LIN {X 0,Y 254.249,Z 344.944,A -85,B 0,C 180,E1 -18935.484,E2 -18935.484} C_VEL
LIN {X 0,Y 252.335,Z 350.692,A -85,B 0,C 180,E1 -18937.788,E2 -18937.788} C_VEL
LIN {X 0,Y 250.743,Z 355.289,A -85,B 0,C 180,E1 -18940.14,E2 -18940.14} C_VEL
LIN {X 0,Y 249.286,Z 359.262,A -85,B 0,C 180,E1 -18942.862,E2 -18942.862} C_VEL
LIN {X 0,Y 248.38,Z 361.475,A -85,B 0,C 180,E1 -18945.022,E2 -18945.022} C_VEL
LIN {X 0,Y 247.644,Z 363.12,A -85,B 0,C 180,E1 -18947.549,E2 -18947.549} C_VEL
LIN {X 0,Y 247.177,Z 363.796,A -85,B 0,C 180,E1 -18950.147,E2 -18950.147} C_VEL
LIN {X 0,Y 246.95,Z 363.273,A -85,B 0,C 180,E1 -18953.299,E2 -18953.299} C_VEL
LIN {X 0,Y 247.021,Z 361.92,A -85,B 0,C 180,E1 -18955.596,E2 -18955.596} C_VEL
LIN {X 0,Y 247.445,Z 359.132,A -85,B 0,C 180,E1 -18958.437,E2 -18958.437} C_VEL
LIN {X 0,Y 248.133,Z 354.726,A -85,B 0,C 180,E1 -18961.405,E2 -18961.405} C_VEL
LIN {X 0,Y 248.912,Z 349.759,A -85,B 0,C 180,E1 -18963.884,E2 -18963.884} C_VEL
LIN {X 0,Y 250.067,Z 343.333,A -85,B 0,C 180,E1 -18966.392,E2 -18966.392} C_VEL
LIN {X 0,Y 251.344,Z 335.987,A -85,B 0,C 180,E1 -18968.685,E2 -18968.685} C_VEL
LIN {X 0,Y 253.013,Z 326.632,A -85,B 0,C 180,E1 -18971.005,E2 -18971.005} C_VEL
LIN {X 0,Y 254.61,Z 316.87,A -85,B 0,C 180,E1 -18972.946,E2 -18972.946} C_VEL
LIN {X 0,Y 256.282,Z 305.858,A -85,B 0,C 180,E1 -18974.696,E2 -18974.696} C_VEL
LIN {X 0,Y 257.875,Z 293.608,A -85,B 0,C 180,E1 -18976.204,E2 -18976.204} C_VEL
LIN {X 0,Y 259.117,Z 281.075,A -85,B 0,C 180,E1 -18977.388,E2 -18977.388} C_VEL
LIN {X 0,Y 260.143,Z 267.516,A -85,B 0,C 180,E1 -18978.285,E2 -18978.285} C_VEL
LIN {X 0,Y 260.78,Z 254.66,A -85,B 0,C 180,E1 -18978.831,E2 -18978.831} C_VEL
LIN {X 0,Y 263.039,Z 190.676,A -85,B 0,C 180,E1 -18980.701,E2 -18980.701} C_VEL
LIN {X 0,Y 258.834,Z 179.431,A -85,B 0,C 180,E1 -18981.466,E2 -18981.466} C_VEL
LIN {X 0,Y 250.247,Z 159.861,A -85,B 0,C 180,E1 -18982.993,E2 -18982.993} C_VEL
LIN {X 0,Y 249.456,Z 157.414,A -85,B 0,C 180,E1 -18983.174,E2 -18983.174} C_VEL
LIN {X 0,Y 249.675,Z 157.384,A -85,B 0,C 180,E1 -18988.387,E2 -18988.387} C_VEL
LIN {X 0,Y 249.675,Z 157.386,A -85,B 0,C 180,E1 -18991.613,E2 -18991.613} C_VEL
LIN {X 0,Y 249.431,Z 157.415,A -85,B 0,C 180,E1 -18996.471,E2 -18996.471} C_VEL
LIN {X 0,Y 249.342,Z 157.425,A -85,B 0,C 180,E1 -18999.736,E2 -18999.736} C_VEL
LIN {X 0,Y 249.175,Z 157.448,A -85,B 0,C 180,E1 -19004.705,E2 -19004.705} C_VEL
LIN {X 0,Y 249.108,Z 157.452,A -85,B 0,C 180,E1 -19008.08,E2 -19008.08} C_VEL
LIN {X 0,Y 249.08,Z 157.456,A -85,B 0,C 180,E1 -19011.519,E2 -19011.519} C_VEL
LIN {X 0,Y 249.117,Z 157.452,A -85,B 0,C 180,E1 -19015.476,E2 -19015.476} C_VEL
LIN {X 0,Y 249.083,Z 157.458,A -85,B 0,C 180,E1 -19018.994,E2 -19018.994} C_VEL
LIN {X 0,Y 249.033,Z 157.465,A -85,B 0,C 180,E1 -19022.425,E2 -19022.425} C_VEL
LIN {X 0,Y 249.056,Z 157.462,A -85,B 0,C 180,E1 -19026.341,E2 -19026.341} C_VEL
LIN {X 0,Y 249.005,Z 157.462,A -85,B 0,C 180,E1 -19030.478,E2 -19030.478} C_VEL
LIN {X 0,Y 249.001,Z 157.467,A -85,B 0,C 180,E1 -19034.879,E2 -19034.879} C_VEL
LIN {X 0,Y 249.015,Z 157.463,A -85,B 0,C 180,E1 -19037.363,E2 -19037.363} C_VEL
LIN {X 0,Y 249.047,Z 157.459,A -85,B 0,C 180,E1 -19042.199,E2 -19042.199} C_VEL
LIN {X 0,Y 249.057,Z 157.461,A -85,B 0,C 180,E1 -19045.642,E2 -19045.642} C_VEL
LIN {X 0,Y 249.047,Z 157.457,A -85,B 0,C 180,E1 -19049.473,E2 -19049.473} C_VEL
LIN {X 0,Y 249.068,Z 157.454,A -85,B 0,C 180,E1 -19053.162,E2 -19053.162} C_VEL
LIN {X 0,Y 249.06,Z 157.459,A -85,B 0,C 180,E1 -19056.731,E2 -19056.731} C_VEL
LIN {X 0,Y 249.108,Z 157.448,A -85,B 0,C 180,E1 -19060.212,E2 -19060.212} C_VEL
LIN {X 0,Y 249.241,Z 157.432,A -85,B 0,C 180,E1 -19063.622,E2 -19063.622} C_VEL
LIN {X 0,Y 249.252,Z 157.435,A -85,B 0,C 180,E1 -19068.617,E2 -19068.617} C_VEL
LIN {X 0,Y 249.481,Z 157.4,A -85,B 0,C 180,E1 -19071.903,E2 -19071.903} C_VEL
LIN {X 0,Y 249.436,Z 157.41,A -85,B 0,C 180,E1 -19076.77,E2 -19076.77} C_VEL
LIN {X 0,Y 249.728,Z 157.373,A -85,B 0,C 180,E1 -19080,E2 -19080} C_VEL
LIN {X 0,Y 249.435,Z 157.406,A -85,B 0,C 180,E1 -19083.231,E2 -19083.231} C_VEL
LIN {X 0,Y 249.479,Z 157.406,A -85,B 0,C 180,E1 -19088.098,E2 -19088.098} C_VEL
LIN {X 0,Y 249.21,Z 157.434,A -85,B 0,C 180,E1 -19092.351,E2 -19092.351} C_VEL
LIN {X 0,Y 248.532,Z 157.522,A -85,B 0,C 180,E1 -19093.701,E2 -19093.701} C_VEL
LIN {X 0,Y 245.64,Z 157.885,A -85,B 0,C 180,E1 -19095.9,E2 -19095.9} C_VEL
LIN {X 0,Y 243.178,Z 158.191,A -85,B 0,C 180,E1 -19097.691,E2 -19097.691} C_VEL
LIN {X 0,Y 242.115,Z 158.322,A -85,B 0,C 180,E1 -19099.081,E2 -19099.081} C_VEL
LIN {X 0,Y 242.025,Z 158.331,A -85,B 0,C 180,E1 -19099.553,E2 -19099.553} C_VEL
LIN {X 0,Y 242.041,Z 158.335,A -85,B 0,C 180,E1 -19103.986,E2 -19103.986} C_VEL
LIN {X 0,Y 242.007,Z 158.336,A -85,B 0,C 180,E1 -19107.688,E2 -19107.688} C_VEL
LIN {X 0,Y 241.977,Z 158.341,A -85,B 0,C 180,E1 -19111.52,E2 -19111.52} C_VEL
LIN {X 0,Y 242.03,Z 158.336,A -85,B 0,C 180,E1 -19115.605,E2 -19115.605} C_VEL
LIN {X 0,Y 241.983,Z 158.342,A -85,B 0,C 180,E1 -19119.714,E2 -19119.714} C_VEL
LIN {X 0,Y 241.939,Z 158.349,A -85,B 0,C 180,E1 -19124.201,E2 -19124.201} C_VEL
LIN {X 0,Y 241.956,Z 158.348,A -85,B 0,C 180,E1 -19128.082,E2 -19128.082} C_VEL
LIN {X 0,Y 242.043,Z 158.414,A -85,B 0,C 180,E1 -19132.281,E2 -19132.281} C_VEL
LIN {X 0,Y 244.127,Z 167.645,A -85,B 0,C 180,E1 -19135.754,E2 -19135.754} C_VEL
LIN {X 0,Y 246.271,Z 177.912,A -85,B 0,C 180,E1 -19139.352,E2 -19139.352} C_VEL
LIN {X 0,Y 249.889,Z 188.242,A -85,B 0,C 180,E1 -19140.086,E2 -19140.086} C_VEL
LIN {X 0,Y 254.57,Z 225.349,A -85,B 0,C 180,E1 -19141.798,E2 -19141.798} C_VEL
LIN {X 0,Y 255.275,Z 233.674,A -85,B 0,C 180,E1 -19142.141,E2 -19142.141} C_VEL
LIN {X 0,Y 253.345,Z 287.616,A -85,B 0,C 180,E1 -19143.816,E2 -19143.816} C_VEL
LIN {X 0,Y 252.151,Z 301.614,A -85,B 0,C 180,E1 -19144.57,E2 -19144.57} C_VEL
LIN {X 0,Y 250.865,Z 313.126,A -85,B 0,C 180,E1 -19145.482,E2 -19145.482} C_VEL
LIN {X 0,Y 249.22,Z 324.982,A -85,B 0,C 180,E1 -19146.747,E2 -19146.747} C_VEL
LIN {X 0,Y 247.383,Z 336.431,A -85,B 0,C 180,E1 -19148.326,E2 -19148.326} C_VEL
LIN {X 0,Y 245.624,Z 346.791,A -85,B 0,C 180,E1 -19150.137,E2 -19150.137} C_VEL
LIN {X 0,Y 243.711,Z 356.55,A -85,B 0,C 180,E1 -19152.285,E2 -19152.285} C_VEL
LIN {X 0,Y 242.748,Z 363.075,A -85,B 0,C 180,E1 -19154.035,E2 -19154.035} C_VEL
LIN {X 0,Y 241.478,Z 370.708,A -85,B 0,C 180,E1 -19156.536,E2 -19156.536} C_VEL
LIN {X 0,Y 240.617,Z 376.823,A -85,B 0,C 180,E1 -19159.056,E2 -19159.056} C_VEL
LIN {X 0,Y 240.174,Z 381.638,A -85,B 0,C 180,E1 -19161.587,E2 -19161.587} C_VEL
LIN {X 0,Y 240.026,Z 385.851,A -85,B 0,C 180,E1 -19164.582,E2 -19164.582} C_VEL
LIN {X 0,Y 240.052,Z 387.865,A -85,B 0,C 180,E1 -19166.643,E2 -19166.643} C_VEL
LIN {X 0,Y 240.072,Z 389.047,A -85,B 0,C 180,E1 -19168.322,E2 -19168.322} C_VEL
LIN {X 0,Y 240.122,Z 389.77,A -85,B 0,C 180,E1 -19170,E2 -19170} C_VEL
LIN {X 0,Y 240.033,Z 390.065,A -85,B 0,C 180,E1 -19171.678,E2 -19171.678} C_VEL
LIN {X 0,Y 239.948,Z 389.962,A -85,B 0,C 180,E1 -19173.358,E2 -19173.358} C_VEL
LIN {X 0,Y 239.882,Z 389.463,A -85,B 0,C 180,E1 -19175.042,E2 -19175.042} C_VEL
LIN {X 0,Y 239.894,Z 388.533,A -85,B 0,C 180,E1 -19176.73,E2 -19176.73} C_VEL
LIN {X 0,Y 240.123,Z 387.193,A -85,B 0,C 180,E1 -19178.415,E2 -19178.415} C_VEL
LIN {X 0,Y 240.68,Z 384.41,A -85,B 0,C 180,E1 -19180.941,E2 -19180.941} C_VEL
LIN {X 0,Y 241.617,Z 380.62,A -85,B 0,C 180,E1 -19183.456,E2 -19183.456} C_VEL
LIN {X 0,Y 243.195,Z 375.731,A -85,B 0,C 180,E1 -19185.934,E2 -19185.934} C_VEL
LIN {X 0,Y 245.131,Z 369.625,A -85,B 0,C 180,E1 -19188.383,E2 -19188.383} C_VEL
LIN {X 0,Y 247.36,Z 362.085,A -85,B 0,C 180,E1 -19190.802,E2 -19190.802} C_VEL
LIN {X 0,Y 249.681,Z 354.448,A -85,B 0,C 180,E1 -19192.77,E2 -19192.77} C_VEL
LIN {X 0,Y 252.469,Z 345.25,A -85,B 0,C 180,E1 -19194.68,E2 -19194.68} C_VEL
LIN {X 0,Y 255.148,Z 335.125,A -85,B 0,C 180,E1 -19196.369,E2 -19196.369} C_VEL
LIN {X 0,Y 257.846,Z 323.973,A -85,B 0,C 180,E1 -19197.824,E2 -19197.824} C_VEL
LIN {X 0,Y 260.362,Z 311.591,A -85,B 0,C 180,E1 -19199.07,E2 -19199.07} C_VEL
LIN {X 0,Y 262.438,Z 299.112,A -85,B 0,C 180,E1 -19199.974,E2 -19199.974} C_VEL
LIN {X 0,Y 263.972,Z 285.064,A -85,B 0,C 180,E1 -19200.686,E2 -19200.686} C_VEL
LIN {X 0,Y 266.579,Z 234.047,A -85,B 0,C 180,E1 -19202.259,E2 -19202.259} C_VEL
LIN {X 0,Y 264.178,Z 213.654,A -85,B 0,C 180,E1 -19203.494,E2 -19203.494} C_VEL
LIN {X 0,Y 262.753,Z 205.326,A -85,B 0,C 180,E1 -19204.097,E2 -19204.097} C_VEL
LIN {X 0,Y 256.837,Z 192.294,A -85,B 0,C 180,E1 -19205.842,E2 -19205.842} C_VEL
LIN {X 0,Y 251.688,Z 182.454,A -85,B 0,C 180,E1 -19207.421,E2 -19207.421} C_VEL
LIN {X 0,Y 249.128,Z 177.872,A -85,B 0,C 180,E1 -19208.251,E2 -19208.251} C_VEL
LIN {X 0,Y 246.506,Z 173.057,A -85,B 0,C 180,E1 -19209.204,E2 -19209.204} C_VEL
LIN {X 0,Y 244.37,Z 165.987,A -85,B 0,C 180,E1 -19212.831,E2 -19212.831} C_VEL
LIN {X 0,Y 241.986,Z 158.344,A -85,B 0,C 180,E1 -19217.362,E2 -19217.362} C_VEL
LIN {X 0,Y 242.019,Z 158.334,A -85,B 0,C 180,E1 -19221.633,E2 -19221.633} C_VEL
LIN {X 0,Y 242.037,Z 158.33,A -85,B 0,C 180,E1 -19224.497,E2 -19224.497} C_VEL
LIN {X 0,Y 241.975,Z 158.344,A -85,B 0,C 180,E1 -19228.48,E2 -19228.48} C_VEL
LIN {X 0,Y 242.002,Z 158.339,A -85,B 0,C 180,E1 -19232.311,E2 -19232.311} C_VEL
LIN {X 0,Y 242.041,Z 158.331,A -85,B 0,C 180,E1 -19236.014,E2 -19236.014} C_VEL
LIN {X 0,Y 242.035,Z 158.332,A -85,B 0,C 180,E1 -19239.607,E2 -19239.607} C_VEL
LIN {X 0,Y 242.163,Z 158.318,A -85,B 0,C 180,E1 -19243.278,E2 -19243.278} C_VEL
LIN {X 0,Y 242.186,Z 158.308,A -85,B 0,C 180,E1 -19248.279,E2 -19248.279} C_VEL
LIN {X 0,Y 242.434,Z 158.28,A -85,B 0,C 180,E1 -19251.665,E2 -19251.665} C_VEL
LIN {X 0,Y 242.26,Z 158.305,A -85,B 0,C 180,E1 -19255.007,E2 -19255.007} C_VEL
LIN {X 0,Y 242.636,Z 158.262,A -85,B 0,C 180,E1 -19258.34,E2 -19258.34} C_VEL
LIN {X 0,Y 242.635,Z 158.262,A -85,B 0,C 180,E1 -19261.659,E2 -19261.659} C_VEL
LIN {X 0,Y 242.421,Z 158.283,A -85,B 0,C 180,E1 -19266.682,E2 -19266.682} C_VEL
LIN {X 0,Y 242.266,Z 158.309,A -85,B 0,C 180,E1 -19270.023,E2 -19270.023} C_VEL
LIN {X 0,Y 242.168,Z 158.323,A -85,B 0,C 180,E1 -19272.784,E2 -19272.784} C_VEL
LIN {X 0,Y 243.206,Z 161.191,A -85,B 0,C 180,E1 -19273.26,E2 -19273.26} C_VEL
LIN {X 0,Y 245.277,Z 163.329,A -85,B 0,C 180,E1 -19273.937,E2 -19273.937} C_VEL
LIN {X 0,Y 247.676,Z 167.09,A -85,B 0,C 180,E1 -19274.747,E2 -19274.747} C_VEL
LIN {X 0,Y 248.99,Z 168.781,A -85,B 0,C 180,E1 -19275.161,E2 -19275.161} C_VEL
LIN {X 0,Y 256.246,Z 179.824,A -85,B 0,C 180,E1 -19277.366,E2 -19277.366} C_VEL
LIN {X 0,Y 263.282,Z 192.025,A -85,B 0,C 180,E1 -19279.347,E2 -19279.347} C_VEL
LIN {X 0,Y 268.227,Z 202.792,A -85,B 0,C 180,E1 -19280.693,E2 -19280.693} C_VEL
LIN {X 0,Y 264.941,Z 262.832,A -85,B 0,C 180,E1 -19282.503,E2 -19282.503} C_VEL
LIN {X 0,Y 263.713,Z 275.612,A -85,B 0,C 180,E1 -19283.164,E2 -19283.164} C_VEL
LIN {X 0,Y 262.155,Z 287.942,A -85,B 0,C 180,E1 -19284.108,E2 -19284.108} C_VEL
LIN {X 0,Y 260.27,Z 299.164,A -85,B 0,C 180,E1 -19285.252,E2 -19285.252} C_VEL
LIN {X 0,Y 257.941,Z 310.086,A -85,B 0,C 180,E1 -19286.674,E2 -19286.674} C_VEL
LIN {X 0,Y 255.21,Z 321.417,A -85,B 0,C 180,E1 -19288.567,E2 -19288.567} C_VEL
LIN {X 0,Y 252.688,Z 330.316,A -85,B 0,C 180,E1 -19290.436,E2 -19290.436} C_VEL
LIN {X 0,Y 250.113,Z 338.389,A -85,B 0,C 180,E1 -19292.545,E2 -19292.545} C_VEL
LIN {X 0,Y 247.851,Z 344.993,A -85,B 0,C 180,E1 -19294.683,E2 -19294.683} C_VEL
LIN {X 0,Y 245.497,Z 351.639,A -85,B 0,C 180,E1 -19297.432,E2 -19297.432} C_VEL
LIN {X 0,Y 243.546,Z 356.786,A -85,B 0,C 180,E1 -19300.266,E2 -19300.266} C_VEL
LIN {X 0,Y 241.941,Z 360.785,A -85,B 0,C 180,E1 -19303.431,E2 -19303.431} C_VEL
LIN {X 0,Y 241.104,Z 362.63,A -85,B 0,C 180,E1 -19305.607,E2 -19305.607} C_VEL
LIN {X 0,Y 240.496,Z 363.763,A -85,B 0,C 180,E1 -19307.769,E2 -19307.769} C_VEL
LIN {X 0,Y 240.12,Z 364.199,A -85,B 0,C 180,E1 -19309.916,E2 -19309.916} C_VEL
LIN {X 0,Y 239.882,Z 363.954,A -85,B 0,C 180,E1 -19312.282,E2 -19312.282} C_VEL
LIN {X 0,Y 239.902,Z 362.595,A -85,B 0,C 180,E1 -19315.111,E2 -19315.111} C_VEL
LIN {X 0,Y 240.298,Z 359.738,A -85,B 0,C 180,E1 -19318.235,E2 -19318.235} C_VEL
LIN {X 0,Y 240.931,Z 355.842,A -85,B 0,C 180,E1 -19321.057,E2 -19321.057} C_VEL
LIN {X 0,Y 241.913,Z 349.852,A -85,B 0,C 180,E1 -19324.166,E2 -19324.166} C_VEL
LIN {X 0,Y 243.185,Z 343.068,A -85,B 0,C 180,E1 -19326.849,E2 -19326.849} C_VEL
LIN {X 0,Y 244.661,Z 334.841,A -85,B 0,C 180,E1 -19329.397,E2 -19329.397} C_VEL
LIN {X 0,Y 246.413,Z 325.395,A -85,B 0,C 180,E1 -19331.716,E2 -19331.716} C_VEL
LIN {X 0,Y 248.089,Z 315.253,A -85,B 0,C 180,E1 -19333.708,E2 -19333.708} C_VEL
LIN {X 0,Y 249.669,Z 304.922,A -85,B 0,C 180,E1 -19335.325,E2 -19335.325} C_VEL
LIN {X 0,Y 251.317,Z 292.397,A -85,B 0,C 180,E1 -19336.867,E2 -19336.867} C_VEL
LIN {X 0,Y 252.543,Z 279.969,A -85,B 0,C 180,E1 -19338.018,E2 -19338.018} C_VEL
LIN {X 0,Y 253.561,Z 266.475,A -85,B 0,C 180,E1 -19338.902,E2 -19338.902} C_VEL
LIN {X 0,Y 254.163,Z 254.123,A -85,B 0,C 180,E1 -19339.416,E2 -19339.416} C_VEL
LIN {X 0,Y 256.396,Z 192.004,A -85,B 0,C 180,E1 -19341.28,E2 -19341.28} C_VEL
LIN {X 0,Y 252.285,Z 181.243,A -85,B 0,C 180,E1 -19342.044,E2 -19342.044} C_VEL
LIN {X 0,Y 244.354,Z 163.164,A -85,B 0,C 180,E1 -19343.505,E2 -19343.505} C_VEL
LIN {X 0,Y 242.467,Z 158.912,A -85,B 0,C 180,E1 -19343.864,E2 -19343.864} C_VEL
LIN {X 0,Y 242.353,Z 158.299,A -85,B 0,C 180,E1 -19343.966,E2 -19343.966} C_VEL
LIN {X 0,Y 242.636,Z 158.261,A -85,B 0,C 180,E1 -19348.34,E2 -19348.34} C_VEL
LIN {X 0,Y 242.635,Z 158.263,A -85,B 0,C 180,E1 -19351.66,E2 -19351.66} C_VEL
LIN {X 0,Y 242.401,Z 158.292,A -85,B 0,C 180,E1 -19356.66,E2 -19356.66} C_VEL
LIN {X 0,Y 242.265,Z 158.306,A -85,B 0,C 180,E1 -19360.024,E2 -19360.024} C_VEL
LIN {X 0,Y 242.134,Z 158.324,A -85,B 0,C 180,E1 -19365.143,E2 -19365.143} C_VEL
LIN {X 0,Y 242.046,Z 158.334,A -85,B 0,C 180,E1 -19368.626,E2 -19368.626} C_VEL
LIN {X 0,Y 242.004,Z 158.338,A -85,B 0,C 180,E1 -19372.181,E2 -19372.181} C_VEL
LIN {X 0,Y 242.066,Z 158.33,A -85,B 0,C 180,E1 -19375.838,E2 -19375.838} C_VEL
LIN {X 0,Y 242.03,Z 158.335,A -85,B 0,C 180,E1 -19379.58,E2 -19379.58} C_VEL
LIN {X 0,Y 241.987,Z 158.34,A -85,B 0,C 180,E1 -19383.491,E2 -19383.491} C_VEL
LIN {X 0,Y 241.99,Z 158.34,A -85,B 0,C 180,E1 -19387.582,E2 -19387.582} C_VEL
LIN {X 0,Y 241.936,Z 158.341,A -85,B 0,C 180,E1 -19391.922,E2 -19391.922} C_VEL
LIN {X 0,Y 241.933,Z 158.347,A -85,B 0,C 180,E1 -19396.571,E2 -19396.571} C_VEL
LIN {X 0,Y 241.956,Z 158.337,A -85,B 0,C 180,E1 -19400.281,E2 -19400.281} C_VEL
LIN {X 0,Y 242.036,Z 158.334,A -85,B 0,C 180,E1 -19404.498,E2 -19404.498} C_VEL
LIN {X 0,Y 241.973,Z 158.337,A -85,B 0,C 180,E1 -19408.48,E2 -19408.48} C_VEL
LIN {X 0,Y 242.001,Z 158.334,A -85,B 0,C 180,E1 -19412.312,E2 -19412.312} C_VEL
LIN {X 0,Y 242.04,Z 158.335,A -85,B 0,C 180,E1 -19416.015,E2 -19416.015} C_VEL
LIN {X 0,Y 242.035,Z 158.332,A -85,B 0,C 180,E1 -19419.608,E2 -19419.608} C_VEL
LIN {X 0,Y 242.163,Z 158.31,A -85,B 0,C 180,E1 -19423.278,E2 -19423.278} C_VEL
LIN {X 0,Y 242.186,Z 158.315,A -85,B 0,C 180,E1 -19428.28,E2 -19428.28} C_VEL
LIN {X 0,Y 242.427,Z 158.279,A -85,B 0,C 180,E1 -19431.666,E2 -19431.666} C_VEL
LIN {X 0,Y 242.26,Z 158.299,A -85,B 0,C 180,E1 -19435.008,E2 -19435.008} C_VEL
LIN {X 0,Y 242.636,Z 158.258,A -85,B 0,C 180,E1 -19438.341,E2 -19438.341} C_VEL
LIN {X 0,Y 242.636,Z 158.254,A -85,B 0,C 180,E1 -19441.66,E2 -19441.66} C_VEL
LIN {X 0,Y 242.431,Z 158.284,A -85,B 0,C 180,E1 -19446.659,E2 -19446.659} C_VEL
LIN {X 0,Y 242.314,Z 158.298,A -85,B 0,C 180,E1 -19450.022,E2 -19450.022} C_VEL
LIN {X 0,Y 242.167,Z 158.319,A -85,B 0,C 180,E1 -19455.141,E2 -19455.141} C_VEL
LIN {X 0,Y 242.073,Z 158.33,A -85,B 0,C 180,E1 -19458.625,E2 -19458.625} C_VEL
LIN {X 0,Y 242.025,Z 158.331,A -85,B 0,C 180,E1 -19459.553,E2 -19459.553} C_VEL
LIN {X 0,Y 241.357,Z 158.418,A -85,B 0,C 180,E1 -19460.941,E2 -19460.941} C_VEL
LIN {X 0,Y 238.537,Z 158.771,A -85,B 0,C 180,E1 -19463.206,E2 -19463.206} C_VEL
LIN {X 0,Y 235.299,Z 159.173,A -85,B 0,C 180,E1 -19466,E2 -19466} C_VEL
LIN {X 0,Y 234.949,Z 159.214,A -85,B 0,C 180,E1 -19466.967,E2 -19466.967} C_VEL
LIN {X 0,Y 234.933,Z 159.221,A -85,B 0,C 180,E1 -19470.568,E2 -19470.568} C_VEL
LIN {X 0,Y 234.961,Z 159.218,A -85,B 0,C 180,E1 -19474.633,E2 -19474.633} C_VEL
LIN {X 0,Y 234.943,Z 159.218,A -85,B 0,C 180,E1 -19478.945,E2 -19478.945} C_VEL
LIN {X 0,Y 234.923,Z 159.221,A -85,B 0,C 180,E1 -19483.478,E2 -19483.478} C_VEL
LIN {X 0,Y 234.923,Z 159.221,A -85,B 0,C 180,E1 -19486.523,E2 -19486.523} C_VEL
LIN {X 0,Y 234.956,Z 159.22,A -85,B 0,C 180,E1 -19491.086,E2 -19491.086} C_VEL
LIN {X 0,Y 235.009,Z 159.336,A -85,B 0,C 180,E1 -19491.727,E2 -19491.727} C_VEL
LIN {X 0,Y 237.011,Z 168.234,A -85,B 0,C 180,E1 -19495.193,E2 -19495.193} C_VEL
LIN {X 0,Y 238.858,Z 177.173,A -85,B 0,C 180,E1 -19498.506,E2 -19498.506} C_VEL
LIN {X 0,Y 243.536,Z 190.303,A -85,B 0,C 180,E1 -19499.507,E2 -19499.507} C_VEL
LIN {X 0,Y 248.087,Z 227.157,A -85,B 0,C 180,E1 -19501.259,E2 -19501.259} C_VEL
LIN {X 0,Y 248.693,Z 233.781,A -85,B 0,C 180,E1 -19501.544,E2 -19501.544} C_VEL
LIN {X 0,Y 246.705,Z 286.78,A -85,B 0,C 180,E1 -19503.227,E2 -19503.227} C_VEL
LIN {X 0,Y 245.666,Z 299.439,A -85,B 0,C 180,E1 -19503.906,E2 -19503.906} C_VEL
LIN {X 0,Y 244.421,Z 310.85,A -85,B 0,C 180,E1 -19504.792,E2 -19504.792} C_VEL
LIN {X 0,Y 242.687,Z 323.235,A -85,B 0,C 180,E1 -19506.082,E2 -19506.082} C_VEL
LIN {X 0,Y 240.698,Z 334.914,A -85,B 0,C 180,E1 -19507.692,E2 -19507.692} C_VEL
LIN {X 0,Y 238.877,Z 345.482,A -85,B 0,C 180,E1 -19509.551,E2 -19509.551} C_VEL
LIN {X 0,Y 237.364,Z 353.754,A -85,B 0,C 180,E1 -19511.349,E2 -19511.349} C_VEL
LIN {X 0,Y 236.414,Z 359.074,A -85,B 0,C 180,E1 -19512.706,E2 -19512.706} C_VEL
LIN {X 0,Y 234.969,Z 367.435,A -85,B 0,C 180,E1 -19515.272,E2 -19515.272} C_VEL
LIN {X 0,Y 233.797,Z 374.134,A -85,B 0,C 180,E1 -19517.853,E2 -19517.853} C_VEL
LIN {X 0,Y 233.243,Z 379.469,A -85,B 0,C 180,E1 -19520.461,E2 -19520.461} C_VEL
LIN {X 0,Y 232.973,Z 383.573,A -85,B 0,C 180,E1 -19523.069,E2 -19523.069} C_VEL
LIN {X 0,Y 232.928,Z 385.674,A -85,B 0,C 180,E1 -19524.807,E2 -19524.807} C_VEL
LIN {X 0,Y 232.965,Z 387.32,A -85,B 0,C 180,E1 -19526.541,E2 -19526.541} C_VEL
LIN {X 0,Y 232.999,Z 388.54,A -85,B 0,C 180,E1 -19528.271,E2 -19528.271} C_VEL
LIN {X 0,Y 233.045,Z 389.327,A -85,B 0,C 180,E1 -19530,E2 -19530} C_VEL
LIN {X 0,Y 232.958,Z 389.656,A -85,B 0,C 180,E1 -19531.729,E2 -19531.729} C_VEL
LIN {X 0,Y 232.788,Z 389.204,A -85,B 0,C 180,E1 -19534.933,E2 -19534.933} C_VEL
LIN {X 0,Y 232.815,Z 388.247,A -85,B 0,C 180,E1 -19536.935,E2 -19536.935} C_VEL
LIN {X 0,Y 233.069,Z 386.941,A -85,B 0,C 180,E1 -19538.671,E2 -19538.671} C_VEL
LIN {X 0,Y 233.949,Z 383.109,A -85,B 0,C 180,E1 -19542.139,E2 -19542.139} C_VEL
LIN {X 0,Y 235.226,Z 379.051,A -85,B 0,C 180,E1 -19544.712,E2 -19544.712} C_VEL
LIN {X 0,Y 237.238,Z 372.898,A -85,B 0,C 180,E1 -19547.677,E2 -19547.677} C_VEL
LIN {X 0,Y 239.252,Z 366.882,A -85,B 0,C 180,E1 -19549.948,E2 -19549.948} C_VEL
LIN {X 0,Y 241.636,Z 359.45,A -85,B 0,C 180,E1 -19552.216,E2 -19552.216} C_VEL
LIN {X 0,Y 244.822,Z 349.56,A -85,B 0,C 180,E1 -19554.598,E2 -19554.598} C_VEL
LIN {X 0,Y 247.938,Z 339.351,A -85,B 0,C 180,E1 -19556.516,E2 -19556.516} C_VEL
LIN {X 0,Y 250.933,Z 327.945,A -85,B 0,C 180,E1 -19558.205,E2 -19558.205} C_VEL
LIN {X 0,Y 253.512,Z 316.836,A -85,B 0,C 180,E1 -19559.477,E2 -19559.477} C_VEL
LIN {X 0,Y 255.882,Z 304.518,A -85,B 0,C 180,E1 -19560.538,E2 -19560.538} C_VEL
LIN {X 0,Y 257.792,Z 290.808,A -85,B 0,C 180,E1 -19561.376,E2 -19561.376} C_VEL
LIN {X 0,Y 258.873,Z 277.464,A -85,B 0,C 180,E1 -19561.91,E2 -19561.91} C_VEL
LIN {X 0,Y 261.098,Z 235.624,A -85,B 0,C 180,E1 -19563.179,E2 -19563.179} C_VEL
LIN {X 0,Y 258.932,Z 216.197,A -85,B 0,C 180,E1 -19564.386,E2 -19564.386} C_VEL
LIN {X 0,Y 257.669,Z 208.41,A -85,B 0,C 180,E1 -19564.973,E2 -19564.973} C_VEL
LIN {X 0,Y 251.967,Z 195.815,A -85,B 0,C 180,E1 -19566.75,E2 -19566.75} C_VEL
LIN {X 0,Y 247.234,Z 186.573,A -85,B 0,C 180,E1 -19568.302,E2 -19568.302} C_VEL
LIN {X 0,Y 244.995,Z 182.575,A -85,B 0,C 180,E1 -19569.065,E2 -19569.065} C_VEL
LIN {X 0,Y 242.061,Z 177.582,A -85,B 0,C 180,E1 -19570.091,E2 -19570.091} C_VEL
LIN {X 0,Y 239.096,Z 172.425,A -85,B 0,C 180,E1 -19571.244,E2 -19571.244} C_VEL
LIN {X 0,Y 237.192,Z 166.322,A -85,B 0,C 180,E1 -19574.673,E2 -19574.673} C_VEL
LIN {X 0,Y 234.931,Z 159.221,A -85,B 0,C 180,E1 -19579.268,E2 -19579.268} C_VEL
LIN {X 0,Y 234.947,Z 159.216,A -85,B 0,C 180,E1 -19583.254,E2 -19583.254} C_VEL
LIN {X 0,Y 234.961,Z 159.21,A -85,B 0,C 180,E1 -19587.424,E2 -19587.424} C_VEL
LIN {X 0,Y 234.937,Z 159.215,A -85,B 0,C 180,E1 -19591.404,E2 -19591.404} C_VEL
LIN {X 0,Y 234.978,Z 159.211,A -85,B 0,C 180,E1 -19595.245,E2 -19595.245} C_VEL
LIN {X 0,Y 234.998,Z 159.208,A -85,B 0,C 180,E1 -19598.968,E2 -19598.968} C_VEL
LIN {X 0,Y 235.096,Z 159.199,A -85,B 0,C 180,E1 -19603.059,E2 -19603.059} C_VEL
LIN {X 0,Y 235.146,Z 159.187,A -85,B 0,C 180,E1 -19607.923,E2 -19607.923} C_VEL
LIN {X 0,Y 235.39,Z 159.16,A -85,B 0,C 180,E1 -19611.414,E2 -19611.414} C_VEL
LIN {X 0,Y 235.405,Z 159.153,A -85,B 0,C 180,E1 -19613.141,E2 -19613.141} C_VEL
LIN {X 0,Y 235.595,Z 159.139,A -85,B 0,C 180,E1 -19618.29,E2 -19618.29} C_VEL
LIN {X 0,Y 235.595,Z 159.139,A -85,B 0,C 180,E1 -19621.709,E2 -19621.709} C_VEL
LIN {X 0,Y 235.372,Z 159.162,A -85,B 0,C 180,E1 -19626.859,E2 -19626.859} C_VEL
LIN {X 0,Y 235.162,Z 159.193,A -85,B 0,C 180,E1 -19630.721,E2 -19630.721} C_VEL
LIN {X 0,Y 236.095,Z 161.954,A -85,B 0,C 180,E1 -19631.189,E2 -19631.189} C_VEL
LIN {X 0,Y 238.223,Z 164.216,A -85,B 0,C 180,E1 -19631.972,E2 -19631.972} C_VEL
LIN {X 0,Y 238.751,Z 164.754,A -85,B 0,C 180,E1 -19632.16,E2 -19632.16} C_VEL
LIN {X 0,Y 240.726,Z 167.985,A -85,B 0,C 180,E1 -19632.916,E2 -19632.916} C_VEL
LIN {X 0,Y 242.201,Z 169.662,A -85,B 0,C 180,E1 -19633.423,E2 -19633.423} C_VEL
LIN {X 0,Y 244.724,Z 173.275,A -85,B 0,C 180,E1 -19634.288,E2 -19634.288} C_VEL
LIN {X 0,Y 251.244,Z 183.366,A -85,B 0,C 180,E1 -19636.401,E2 -19636.401} C_VEL
LIN {X 0,Y 257.758,Z 194.486,A -85,B 0,C 180,E1 -19638.329,E2 -19638.329} C_VEL
LIN {X 0,Y 262.537,Z 204.672,A -85,B 0,C 180,E1 -19639.722,E2 -19639.722} C_VEL
LIN {X 0,Y 262.624,Z 206.578,A -85,B 0,C 180,E1 -19639.816,E2 -19639.816} C_VEL
LIN {X 0,Y 259.317,Z 263.806,A -85,B 0,C 180,E1 -19641.575,E2 -19641.575} C_VEL
LIN {X 0,Y 257.93,Z 277.288,A -85,B 0,C 180,E1 -19642.301,E2 -19642.301} C_VEL
LIN {X 0,Y 256.165,Z 290.056,A -85,B 0,C 180,E1 -19643.334,E2 -19643.334} C_VEL
LIN {X 0,Y 253.854,Z 302.502,A -85,B 0,C 180,E1 -19644.698,E2 -19644.698} C_VEL
LIN {X 0,Y 251.49,Z 312.773,A -85,B 0,C 180,E1 -19646.137,E2 -19646.137} C_VEL
LIN {X 0,Y 248.745,Z 323.234,A -85,B 0,C 180,E1 -19648.003,E2 -19648.003} C_VEL
LIN {X 0,Y 245.817,Z 332.731,A -85,B 0,C 180,E1 -19650.134,E2 -19650.134} C_VEL
LIN {X 0,Y 243.185,Z 340.459,A -85,B 0,C 180,E1 -19652.295,E2 -19652.295} C_VEL
LIN {X 0,Y 241.074,Z 346.183,A -85,B 0,C 180,E1 -19654.267,E2 -19654.267} C_VEL
LIN {X 0,Y 238.987,Z 351.644,A -85,B 0,C 180,E1 -19656.593,E2 -19656.593} C_VEL
LIN {X 0,Y 236.898,Z 356.942,A -85,B 0,C 180,E1 -19659.527,E2 -19659.527} C_VEL
LIN {X 0,Y 235.619,Z 359.943,A -85,B 0,C 180,E1 -19661.782,E2 -19661.782} C_VEL
LIN {X 0,Y 234.566,Z 362.16,A -85,B 0,C 180,E1 -19664.022,E2 -19664.022} C_VEL
LIN {X 0,Y 233.805,Z 363.672,A -85,B 0,C 180,E1 -19666.262,E2 -19666.262} C_VEL
LIN {X 0,Y 233.194,Z 364.542,A -85,B 0,C 180,E1 -19668.89,E2 -19668.89} C_VEL
LIN {X 0,Y 232.835,Z 364.459,A -85,B 0,C 180,E1 -19671.701,E2 -19671.701} C_VEL
LIN {X 0,Y 232.823,Z 362.988,A -85,B 0,C 180,E1 -19675.003,E2 -19675.003} C_VEL
LIN {X 0,Y 233.088,Z 360.807,A -85,B 0,C 180,E1 -19677.591,E2 -19677.591} C_VEL
LIN {X 0,Y 233.74,Z 356.883,A -85,B 0,C 180,E1 -19680.687,E2 -19680.687} C_VEL
LIN {X 0,Y 234.491,Z 352.387,A -85,B 0,C 180,E1 -19683.284,E2 -19683.284} C_VEL
LIN {X 0,Y 235.739,Z 345.647,A -85,B 0,C 180,E1 -19686.268,E2 -19686.268} C_VEL
LIN {X 0,Y 237.081,Z 338.583,A -85,B 0,C 180,E1 -19688.707,E2 -19688.707} C_VEL
LIN {X 0,Y 238.709,Z 329.948,A -85,B 0,C 180,E1 -19691.104,E2 -19691.104} C_VEL
LIN {X 0,Y 240.491,Z 320.073,A -85,B 0,C 180,E1 -19693.298,E2 -19693.298} C_VEL
LIN {X 0,Y 242.173,Z 310.035,A -85,B 0,C 180,E1 -19695.075,E2 -19695.075} C_VEL
LIN {X 0,Y 243.926,Z 297.815,A -85,B 0,C 180,E1 -19696.793,E2 -19696.793} C_VEL
LIN {X 0,Y 245.231,Z 286.652,A -85,B 0,C 180,E1 -19698.006,E2 -19698.006} C_VEL
LIN {X 0,Y 246.451,Z 273.487,A -85,B 0,C 180,E1 -19699.058,E2 -19699.058} C_VEL
LIN {X 0,Y 247.285,Z 260.459,A -85,B 0,C 180,E1 -19699.768,E2 -19699.768} C_VEL
LIN {X 0,Y 249.818,Z 193.519,A -85,B 0,C 180,E1 -19701.865,E2 -19701.865} C_VEL
LIN {X 0,Y 245.262,Z 181.895,A -85,B 0,C 180,E1 -19702.74,E2 -19702.74} C_VEL
LIN {X 0,Y 237.732,Z 164.86,A -85,B 0,C 180,E1 -19704.182,E2 -19704.182} C_VEL
LIN {X 0,Y 235.445,Z 160.207,A -85,B 0,C 180,E1 -19704.621,E2 -19704.621} C_VEL
LIN {X 0,Y 235.257,Z 159.182,A -85,B 0,C 180,E1 -19704.713,E2 -19704.713} C_VEL
LIN {X 0,Y 235.595,Z 159.138,A -85,B 0,C 180,E1 -19708.291,E2 -19708.291} C_VEL
LIN {X 0,Y 235.594,Z 159.14,A -85,B 0,C 180,E1 -19711.71,E2 -19711.71} C_VEL
LIN {X 0,Y 235.351,Z 159.171,A -85,B 0,C 180,E1 -19716.86,E2 -19716.86} C_VEL
LIN {X 0,Y 235.211,Z 159.186,A -85,B 0,C 180,E1 -19720.328,E2 -19720.328} C_VEL
LIN {X 0,Y 235.079,Z 159.201,A -85,B 0,C 180,E1 -19725.609,E2 -19725.609} C_VEL
LIN {X 0,Y 234.987,Z 159.214,A -85,B 0,C 180,E1 -19729.207,E2 -19729.207} C_VEL
LIN {X 0,Y 234.951,Z 159.219,A -85,B 0,C 180,E1 -19732.884,E2 -19732.884} C_VEL
LIN {X 0,Y 234.969,Z 159.217,A -85,B 0,C 180,E1 -19736.657,E2 -19736.657} C_VEL
LIN {X 0,Y 234.931,Z 159.221,A -85,B 0,C 180,E1 -19740.568,E2 -19740.568} C_VEL
LIN {X 0,Y 234.941,Z 159.219,A -85,B 0,C 180,E1 -19744.636,E2 -19744.636} C_VEL
LIN {X 0,Y 234.941,Z 159.216,A -85,B 0,C 180,E1 -19748.944,E2 -19748.944} C_VEL
LIN {X 0,Y 234.886,Z 159.222,A -85,B 0,C 180,E1 -19753.486,E2 -19753.486} C_VEL
LIN {X 0,Y 234.886,Z 159.225,A -85,B 0,C 180,E1 -19756.514,E2 -19756.514} C_VEL
LIN {X 0,Y 234.919,Z 159.212,A -85,B 0,C 180,E1 -19761.079,E2 -19761.079} C_VEL
LIN {X 0,Y 234.959,Z 159.215,A -85,B 0,C 180,E1 -19765.367,E2 -19765.367} C_VEL
LIN {X 0,Y 234.922,Z 159.216,A -85,B 0,C 180,E1 -19769.431,E2 -19769.431} C_VEL
LIN {X 0,Y 234.993,Z 159.211,A -85,B 0,C 180,E1 -19773.794,E2 -19773.794} C_VEL
LIN {X 0,Y 234.997,Z 159.209,A -85,B 0,C 180,E1 -19778.969,E2 -19778.969} C_VEL
LIN {X 0,Y 235.096,Z 159.188,A -85,B 0,C 180,E1 -19783.06,E2 -19783.06} C_VEL
LIN {X 0,Y 235.146,Z 159.192,A -85,B 0,C 180,E1 -19787.924,E2 -19787.924} C_VEL
LIN {X 0,Y 235.377,Z 159.158,A -85,B 0,C 180,E1 -19791.414,E2 -19791.414} C_VEL
LIN {X 0,Y 235.404,Z 159.151,A -85,B 0,C 180,E1 -19793.142,E2 -19793.142} C_VEL
LIN {X 0,Y 235.596,Z 159.134,A -85,B 0,C 180,E1 -19798.291,E2 -19798.291} C_VEL
LIN {X 0,Y 235.595,Z 159.13,A -85,B 0,C 180,E1 -19801.71,E2 -19801.71} C_VEL
LIN {X 0,Y 235.402,Z 159.16,A -85,B 0,C 180,E1 -19806.859,E2 -19806.859} C_VEL
LIN {X 0,Y 235.238,Z 159.18,A -85,B 0,C 180,E1 -19810.327,E2 -19810.327} C_VEL
LIN {X 0,Y 235.114,Z 159.196,A -85,B 0,C 180,E1 -19815.607,E2 -19815.607} C_VEL
LIN {X 0,Y 234.989,Z 159.207,A -85,B 0,C 180,E1 -19819.534,E2 -19819.534} C_VEL
LIN {X 0,Y 234.953,Z 159.218,A -85,B 0,C 180,E1 -19822.884,E2 -19822.884} C_VEL
LIN {X 0,Y 234.949,Z 159.214,A -85,B 0,C 180,E1 -19826.967,E2 -19826.967} C_VEL
LIN {X 0,Y 234.232,Z 159.309,A -85,B 0,C 180,E1 -19828.397,E2 -19828.397} C_VEL
LIN {X 0,Y 231.369,Z 159.664,A -85,B 0,C 180,E1 -19830.732,E2 -19830.732} C_VEL
LIN {X 0,Y 228.966,Z 159.964,A -85,B 0,C 180,E1 -19832.635,E2 -19832.635} C_VEL
LIN {X 0,Y 227.94,Z 160.094,A -85,B 0,C 180,E1 -19834.111,E2 -19834.111} C_VEL
LIN {X 0,Y 227.856,Z 160.097,A -85,B 0,C 180,E1 -19834.612,E2 -19834.612} C_VEL
LIN {X 0,Y 227.872,Z 160.102,A -85,B 0,C 180,E1 -19838.086,E2 -19838.086} C_VEL
LIN {X 0,Y 227.865,Z 160.1,A -85,B 0,C 180,E1 -19842.73,E2 -19842.73} C_VEL
LIN {X 0,Y 227.869,Z 160.102,A -85,B 0,C 180,E1 -19847.75,E2 -19847.75} C_VEL
LIN {X 0,Y 227.912,Z 160.105,A -85,B 0,C 180,E1 -19851.084,E2 -19851.084} C_VEL
LIN {X 0,Y 229.831,Z 168.517,A -85,B 0,C 180,E1 -19854.479,E2 -19854.479} C_VEL
LIN {X 0,Y 231.623,Z 176.956,A -85,B 0,C 180,E1 -19857.685,E2 -19857.685} C_VEL
LIN {X 0,Y 237.176,Z 192.061,A -85,B 0,C 180,E1 -19858.881,E2 -19858.881} C_VEL
LIN {X 0,Y 241.567,Z 228.173,A -85,B 0,C 180,E1 -19860.658,E2 -19860.658} C_VEL
LIN {X 0,Y 242.091,Z 234.591,A -85,B 0,C 180,E1 -19860.938,E2 -19860.938} C_VEL
LIN {X 0,Y 240.048,Z 287.005,A -85,B 0,C 180,E1 -19862.659,E2 -19862.659} C_VEL
LIN {X 0,Y 238.974,Z 299.463,A -85,B 0,C 180,E1 -19863.353,E2 -19863.353} C_VEL
LIN {X 0,Y 237.537,Z 311.88,A -85,B 0,C 180,E1 -19864.36,E2 -19864.36} C_VEL
LIN {X 0,Y 235.911,Z 323.072,A -85,B 0,C 180,E1 -19865.585,E2 -19865.585} C_VEL
LIN {X 0,Y 233.858,Z 334.706,A -85,B 0,C 180,E1 -19867.237,E2 -19867.237} C_VEL
LIN {X 0,Y 231.989,Z 345.248,A -85,B 0,C 180,E1 -19869.148,E2 -19869.148} C_VEL
LIN {X 0,Y 230.393,Z 353.607,A -85,B 0,C 180,E1 -19871.022,E2 -19871.022} C_VEL
LIN {X 0,Y 229.527,Z 358.021,A -85,B 0,C 180,E1 -19872.17,E2 -19872.17} C_VEL
LIN {X 0,Y 228.06,Z 366.513,A -85,B 0,C 180,E1 -19874.815,E2 -19874.815} C_VEL
LIN {X 0,Y 226.813,Z 373.309,A -85,B 0,C 180,E1 -19877.473,E2 -19877.473} C_VEL
LIN {X 0,Y 226.211,Z 378.733,A -85,B 0,C 180,E1 -19880.161,E2 -19880.161} C_VEL
LIN {X 0,Y 225.904,Z 382.918,A -85,B 0,C 180,E1 -19882.851,E2 -19882.851} C_VEL
LIN {X 0,Y 225.884,Z 385.096,A -85,B 0,C 180,E1 -19884.644,E2 -19884.644} C_VEL
LIN {X 0,Y 225.88,Z 386.776,A -85,B 0,C 180,E1 -19886.432,E2 -19886.432} C_VEL
LIN {X 0,Y 225.927,Z 388.031,A -85,B 0,C 180,E1 -19888.217,E2 -19888.217} C_VEL
LIN {X 0,Y 225.969,Z 388.869,A -85,B 0,C 180,E1 -19890,E2 -19890} C_VEL
LIN {X 0,Y 225.884,Z 389.247,A -85,B 0,C 180,E1 -19891.783,E2 -19891.783} C_VEL
LIN {X 0,Y 225.717,Z 388.926,A -85,B 0,C 180,E1 -19894.882,E2 -19894.882} C_VEL
LIN {X 0,Y 225.761,Z 387.948,A -85,B 0,C 180,E1 -19897.153,E2 -19897.153} C_VEL
LIN {X 0,Y 226.012,Z 386.705,A -85,B 0,C 180,E1 -19898.944,E2 -19898.944} C_VEL
LIN {X 0,Y 226.663,Z 384.072,A -85,B 0,C 180,E1 -19901.627,E2 -19901.627} C_VEL
LIN {X 0,Y 227.796,Z 380.442,A -85,B 0,C 180,E1 -19904.289,E2 -19904.289} C_VEL
LIN {X 0,Y 229.534,Z 375.74,A -85,B 0,C 180,E1 -19906.91,E2 -19906.91} C_VEL
LIN {X 0,Y 232.098,Z 368.578,A -85,B 0,C 180,E1 -19909.961,E2 -19909.961} C_VEL
LIN {X 0,Y 234.609,Z 361.142,A -85,B 0,C 180,E1 -19912.454,E2 -19912.454} C_VEL
LIN {X 0,Y 237.268,Z 353.508,A -85,B 0,C 180,E1 -19914.499,E2 -19914.499} C_VEL
LIN {X 0,Y 240.351,Z 344.318,A -85,B 0,C 180,E1 -19916.482,E2 -19916.482} C_VEL
LIN {X 0,Y 243.651,Z 332.926,A -85,B 0,C 180,E1 -19918.42,E2 -19918.42} C_VEL
LIN {X 0,Y 246.674,Z 321.511,A -85,B 0,C 180,E1 -19919.907,E2 -19919.907} C_VEL
LIN {X 0,Y 249.211,Z 309.706,A -85,B 0,C 180,E1 -19921.093,E2 -19921.093} C_VEL
LIN {X 0,Y 251.509,Z 296.161,A -85,B 0,C 180,E1 -19922.068,E2 -19922.068} C_VEL
LIN {X 0,Y 252.961,Z 283.161,A -85,B 0,C 180,E1 -19922.715,E2 -19922.715} C_VEL
LIN {X 0,Y 255.662,Z 236.407,A -85,B 0,C 180,E1 -19924.187,E2 -19924.187} C_VEL
LIN {X 0,Y 253.701,Z 217.879,A -85,B 0,C 180,E1 -19925.39,E2 -19925.39} C_VEL
LIN {X 0,Y 252.681,Z 211.613,A -85,B 0,C 180,E1 -19925.886,E2 -19925.886} C_VEL
LIN {X 0,Y 247.546,Z 200.024,A -85,B 0,C 180,E1 -19927.583,E2 -19927.583} C_VEL
LIN {X 0,Y 241.898,Z 188.729,A -85,B 0,C 180,E1 -19929.57,E2 -19929.57} C_VEL
LIN {X 0,Y 238.229,Z 182.499,A -85,B 0,C 180,E1 -19930.916,E2 -19930.916} C_VEL
LIN {X 0,Y 235.004,Z 177.198,A -85,B 0,C 180,E1 -19932.179,E2 -19932.179} C_VEL
LIN {X 0,Y 231.873,Z 172.315,A -85,B 0,C 180,E1 -19933.476,E2 -19933.476} C_VEL
LIN {X 0,Y 231.525,Z 171.354,A -85,B 0,C 180,E1 -19933.827,E2 -19933.827} C_VEL
LIN {X 0,Y 229.592,Z 165.323,A -85,B 0,C 180,E1 -19937.667,E2 -19937.667} C_VEL
LIN {X 0,Y 227.888,Z 160.093,A -85,B 0,C 180,E1 -19941.501,E2 -19941.501} C_VEL
LIN {X 0,Y 227.902,Z 160.09,A -85,B 0,C 180,E1 -19944.132,E2 -19944.132} C_VEL
LIN {X 0,Y 227.87,Z 160.099,A -85,B 0,C 180,E1 -19948.377,E2 -19948.377} C_VEL
LIN {X 0,Y 227.879,Z 160.098,A -85,B 0,C 180,E1 -19952.444,E2 -19952.444} C_VEL
LIN {X 0,Y 227.906,Z 160.088,A -85,B 0,C 180,E1 -19956.366,E2 -19956.366} C_VEL
LIN {X 0,Y 227.937,Z 160.083,A -85,B 0,C 180,E1 -19960.174,E2 -19960.174} C_VEL
LIN {X 0,Y 228.057,Z 160.069,A -85,B 0,C 180,E1 -19963.897,E2 -19963.897} C_VEL
LIN {X 0,Y 228.171,Z 160.054,A -85,B 0,C 180,E1 -19969.35,E2 -19969.35} C_VEL
LIN {X 0,Y 228.357,Z 160.03,A -85,B 0,C 180,E1 -19972.928,E2 -19972.928} C_VEL
LIN {X 0,Y 228.554,Z 160.016,A -85,B 0,C 180,E1 -19978.238,E2 -19978.238} C_VEL
LIN {X 0,Y 228.554,Z 160.015,A -85,B 0,C 180,E1 -19981.762,E2 -19981.762} C_VEL
LIN {X 0,Y 228.292,Z 160.046,A -85,B 0,C 180,E1 -19988.185,E2 -19988.185} C_VEL
LIN {X 0,Y 228.322,Z 160.311,A -85,B 0,C 180,E1 -19988.407,E2 -19988.407} C_VEL
LIN {X 0,Y 229.322,Z 162.991,A -85,B 0,C 180,E1 -19988.948,E2 -19988.948} C_VEL
LIN {X 0,Y 231.537,Z 165.226,A -85,B 0,C 180,E1 -19989.877,E2 -19989.877} C_VEL
LIN {X 0,Y 234.164,Z 169.266,A -85,B 0,C 180,E1 -19990.992,E2 -19990.992} C_VEL
LIN {X 0,Y 235.614,Z 170.862,A -85,B 0,C 180,E1 -19991.54,E2 -19991.54} C_VEL
LIN {X 0,Y 238.167,Z 174.466,A -85,B 0,C 180,E1 -19992.515,E2 -19992.515} C_VEL
LIN {X 0,Y 244.064,Z 183.085,A -85,B 0,C 180,E1 -19994.603,E2 -19994.603} C_VEL
LIN {X 0,Y 250.546,Z 193.959,A -85,B 0,C 180,E1 -19996.732,E2 -19996.732} C_VEL
LIN {X 0,Y 255.131,Z 202.569,A -85,B 0,C 180,E1 -19998.126,E2 -19998.126} C_VEL
LIN {X 0,Y 257.289,Z 207.676,A -85,B 0,C 180,E1 -19998.799,E2 -19998.799} C_VEL
LIN {X 0,Y 253.828,Z 264.233,A -85,B 0,C 180,E1 -20000.577,E2 -20000.577} C_VEL
LIN {X 0,Y 252.392,Z 277.535,A -85,B 0,C 180,E1 -20001.305,E2 -20001.305} C_VEL
LIN {X 0,Y 250.654,Z 289.711,A -85,B 0,C 180,E1 -20002.291,E2 -20002.291} C_VEL
LIN {X 0,Y 248.197,Z 302.495,A -85,B 0,C 180,E1 -20003.699,E2 -20003.699} C_VEL
LIN {X 0,Y 245.419,Z 313.995,A -85,B 0,C 180,E1 -20005.339,E2 -20005.339} C_VEL
LIN {X 0,Y 242.563,Z 324.176,A -85,B 0,C 180,E1 -20007.218,E2 -20007.218} C_VEL
LIN {X 0,Y 239.412,Z 333.892,A -85,B 0,C 180,E1 -20009.473,E2 -20009.473} C_VEL
LIN {X 0,Y 236.574,Z 341.705,A -85,B 0,C 180,E1 -20011.76,E2 -20011.76} C_VEL
LIN {X 0,Y 234.065,Z 348.081,A -85,B 0,C 180,E1 -20014.111,E2 -20014.111} C_VEL
LIN {X 0,Y 231.913,Z 353.251,A -85,B 0,C 180,E1 -20016.503,E2 -20016.503} C_VEL
LIN {X 0,Y 230.184,Z 357.282,A -85,B 0,C 180,E1 -20018.872,E2 -20018.872} C_VEL
LIN {X 0,Y 228.238,Z 361.513,A -85,B 0,C 180,E1 -20022.353,E2 -20022.353} C_VEL
LIN {X 0,Y 226.967,Z 363.832,A -85,B 0,C 180,E1 -20025.413,E2 -20025.413} C_VEL
LIN {X 0,Y 226.251,Z 364.866,A -85,B 0,C 180,E1 -20028.202,E2 -20028.202} C_VEL
LIN {X 0,Y 225.771,Z 364.854,A -85,B 0,C 180,E1 -20031.496,E2 -20031.496} C_VEL
LIN {X 0,Y 225.669,Z 363.868,A -85,B 0,C 180,E1 -20034.068,E2 -20034.068} C_VEL
LIN {X 0,Y 225.928,Z 361.621,A -85,B 0,C 180,E1 -20037.128,E2 -20037.128} C_VEL
LIN {X 0,Y 226.548,Z 357.914,A -85,B 0,C 180,E1 -20040.298,E2 -20040.298} C_VEL
LIN {X 0,Y 227.293,Z 353.464,A -85,B 0,C 180,E1 -20043.053,E2 -20043.053} C_VEL
LIN {X 0,Y 228.426,Z 347.374,A -85,B 0,C 180,E1 -20045.942,E2 -20045.942} C_VEL
LIN {X 0,Y 229.759,Z 340.633,A -85,B 0,C 180,E1 -20048.466,E2 -20048.466} C_VEL
LIN {X 0,Y 231.455,Z 332.244,A -85,B 0,C 180,E1 -20050.971,E2 -20050.971} C_VEL
LIN {X 0,Y 233.272,Z 322.496,A -85,B 0,C 180,E1 -20053.295,E2 -20053.295} C_VEL
LIN {X 0,Y 235.121,Z 312.067,A -85,B 0,C 180,E1 -20055.282,E2 -20055.282} C_VEL
LIN {X 0,Y 236.851,Z 300.83,A -85,B 0,C 180,E1 -20056.967,E2 -20056.967} C_VEL
LIN {X 0,Y 238.428,Z 288.401,A -85,B 0,C 180,E1 -20058.416,E2 -20058.416} C_VEL
LIN {X 0,Y 239.558,Z 276.805,A -85,B 0,C 180,E1 -20059.435,E2 -20059.435} C_VEL
LIN {X 0,Y 240.545,Z 263.196,A -85,B 0,C 180,E1 -20060.254,E2 -20060.254} C_VEL
LIN {X 0,Y 241.516,Z 241.207,A -85,B 0,C 180,E1 -20061.017,E2 -20061.017} C_VEL
LIN {X 0,Y 243.312,Z 195.172,A -85,B 0,C 180,E1 -20062.472,E2 -20062.472} C_VEL
LIN {X 0,Y 235.098,Z 175.135,A -85,B 0,C 180,E1 -20064.102,E2 -20064.102} C_VEL
LIN {X 0,Y 228.345,Z 160.853,A -85,B 0,C 180,E1 -20065.449,E2 -20065.449} C_VEL
LIN {X 0,Y 228.199,Z 160.059,A -85,B 0,C 180,E1 -20065.584,E2 -20065.584} C_VEL
LIN {X 0,Y 228.554,Z 160.015,A -85,B 0,C 180,E1 -20068.238,E2 -20068.238} C_VEL
LIN {X 0,Y 228.553,Z 160.017,A -85,B 0,C 180,E1 -20071.762,E2 -20071.762} C_VEL
LIN {X 0,Y 228.303,Z 160.05,A -85,B 0,C 180,E1 -20077.073,E2 -20077.073} C_VEL
LIN {X 0,Y 228.142,Z 160.067,A -85,B 0,C 180,E1 -20080.651,E2 -20080.651} C_VEL
LIN {X 0,Y 228.037,Z 160.079,A -85,B 0,C 180,E1 -20084.274,E2 -20084.274} C_VEL
LIN {X 0,Y 227.953,Z 160.087,A -85,B 0,C 180,E1 -20087.957,E2 -20087.957} C_VEL
LIN {X 0,Y 227.915,Z 160.093,A -85,B 0,C 180,E1 -20092.32,E2 -20092.32} C_VEL
LIN {X 0,Y 227.942,Z 160.092,A -85,B 0,C 180,E1 -20096.603,E2 -20096.603} C_VEL
LIN {X 0,Y 227.908,Z 160.096,A -85,B 0,C 180,E1 -20100.296,E2 -20100.296} C_VEL
LIN {X 0,Y 227.88,Z 160.098,A -85,B 0,C 180,E1 -20103.72,E2 -20103.72} C_VEL
LIN {X 0,Y 227.843,Z 160.104,A -85,B 0,C 180,E1 -20108.091,E2 -20108.091} C_VEL
LIN {X 0,Y 227.81,Z 160.105,A -85,B 0,C 180,E1 -20112.742,E2 -20112.742} C_VEL
LIN {X 0,Y 227.81,Z 160.105,A -85,B 0,C 180,E1 -20117.258,E2 -20117.258} C_VEL
LIN {X 0,Y 227.847,Z 160.096,A -85,B 0,C 180,E1 -20121.91,E2 -20121.91} C_VEL
LIN {X 0,Y 227.887,Z 160.097,A -85,B 0,C 180,E1 -20126.282,E2 -20126.282} C_VEL
LIN {X 0,Y 227.903,Z 160.081,A -85,B 0,C 180,E1 -20130.436,E2 -20130.436} C_VEL
LIN {X 0,Y 227.924,Z 160.091,A -85,B 0,C 180,E1 -20134.426,E2 -20134.426} C_VEL
LIN {X 0,Y 227.947,Z 160.087,A -85,B 0,C 180,E1 -20138.286,E2 -20138.286} C_VEL
LIN {X 0,Y 228.034,Z 160.066,A -85,B 0,C 180,E1 -20142.826,E2 -20142.826} C_VEL
LIN {X 0,Y 228.093,Z 160.073,A -85,B 0,C 180,E1 -20147.545,E2 -20147.545} C_VEL
LIN {X 0,Y 228.306,Z 160.041,A -85,B 0,C 180,E1 -20151.146,E2 -20151.146} C_VEL
LIN {X 0,Y 228.355,Z 160.029,A -85,B 0,C 180,E1 -20152.929,E2 -20152.929} C_VEL
LIN {X 0,Y 228.554,Z 160.011,A -85,B 0,C 180,E1 -20158.238,E2 -20158.238} C_VEL
LIN {X 0,Y 228.554,Z 160.007,A -85,B 0,C 180,E1 -20161.762,E2 -20161.762} C_VEL
LIN {X 0,Y 228.353,Z 160.04,A -85,B 0,C 180,E1 -20167.072,E2 -20167.072} C_VEL
LIN {X 0,Y 228.163,Z 160.061,A -85,B 0,C 180,E1 -20170.651,E2 -20170.651} C_VEL
LIN {X 0,Y 228.065,Z 160.071,A -85,B 0,C 180,E1 -20174.272,E2 -20174.272} C_VEL
LIN {X 0,Y 228.003,Z 160.082,A -85,B 0,C 180,E1 -20177.954,E2 -20177.954} C_VEL
LIN {X 0,Y 227.917,Z 160.093,A -85,B 0,C 180,E1 -20182.321,E2 -20182.321} C_VEL
LIN {X 0,Y 227.916,Z 160.09,A -85,B 0,C 180,E1 -20186.937,E2 -20186.937} C_VEL
LIN {X 0,Y 227.91,Z 160.098,A -85,B 0,C 180,E1 -20190.297,E2 -20190.297} C_VEL
LIN {X 0,Y 227.856,Z 160.097,A -85,B 0,C 180,E1 -20194.612,E2 -20194.612} C_VEL
LIN {X 0,Y 227.184,Z 160.188,A -85,B 0,C 180,E1 -20196.088,E2 -20196.088} C_VEL
LIN {X 0,Y 224.322,Z 160.542,A -85,B 0,C 180,E1 -20198.497,E2 -20198.497} C_VEL
LIN {X 0,Y 221.905,Z 160.844,A -85,B 0,C 180,E1 -20200.462,E2 -20200.462} C_VEL
LIN {X 0,Y 220.888,Z 160.971,A -85,B 0,C 180,E1 -20201.988,E2 -20201.988} C_VEL
LIN {X 0,Y 220.816,Z 160.978,A -85,B 0,C 180,E1 -20202.506,E2 -20202.506} C_VEL
LIN {X 0,Y 220.831,Z 160.976,A -85,B 0,C 180,E1 -20207.053,E2 -20207.053} C_VEL
LIN {X 0,Y 220.823,Z 161.031,A -85,B 0,C 180,E1 -20210.467,E2 -20210.467} C_VEL
LIN {X 0,Y 222.91,Z 169.866,A -85,B 0,C 180,E1 -20214.17,E2 -20214.17} C_VEL
LIN {X 0,Y 224.304,Z 176.41,A -85,B 0,C 180,E1 -20216.778,E2 -20216.778} C_VEL
LIN {X 0,Y 230.874,Z 194.374,A -85,B 0,C 180,E1 -20218.261,E2 -20218.261} C_VEL
LIN {X 0,Y 234.932,Z 227.849,A -85,B 0,C 180,E1 -20219.961,E2 -20219.961} C_VEL
LIN {X 0,Y 235.511,Z 235.807,A -85,B 0,C 180,E1 -20220.315,E2 -20220.315} C_VEL
LIN {X 0,Y 233.469,Z 286.132,A -85,B 0,C 180,E1 -20222.004,E2 -20222.004} C_VEL
LIN {X 0,Y 232.475,Z 298.013,A -85,B 0,C 180,E1 -20222.669,E2 -20222.669} C_VEL
LIN {X 0,Y 230.994,Z 310.694,A -85,B 0,C 180,E1 -20223.701,E2 -20223.701} C_VEL
LIN {X 0,Y 229.15,Z 322.904,A -85,B 0,C 180,E1 -20225.057,E2 -20225.057} C_VEL
LIN {X 0,Y 227.377,Z 333.22,A -85,B 0,C 180,E1 -20226.55,E2 -20226.55} C_VEL
LIN {X 0,Y 225.273,Z 343.917,A -85,B 0,C 180,E1 -20228.496,E2 -20228.496} C_VEL
LIN {X 0,Y 223.417,Z 353.489,A -85,B 0,C 180,E1 -20230.685,E2 -20230.685} C_VEL
LIN {X 0,Y 221.925,Z 361.522,A -85,B 0,C 180,E1 -20232.966,E2 -20232.966} C_VEL
LIN {X 0,Y 220.491,Z 369.227,A -85,B 0,C 180,E1 -20235.698,E2 -20235.698} C_VEL
LIN {X 0,Y 219.343,Z 376.32,A -85,B 0,C 180,E1 -20238.916,E2 -20238.916} C_VEL
LIN {X 0,Y 218.914,Z 380.988,A -85,B 0,C 180,E1 -20241.694,E2 -20241.694} C_VEL
LIN {X 0,Y 218.8,Z 384.747,A -85,B 0,C 180,E1 -20244.714,E2 -20244.714} C_VEL
LIN {X 0,Y 218.8,Z 386.225,A -85,B 0,C 180,E1 -20246.317,E2 -20246.317} C_VEL
LIN {X 0,Y 218.856,Z 387.516,A -85,B 0,C 180,E1 -20248.16,E2 -20248.16} C_VEL
LIN {X 0,Y 218.896,Z 388.389,A -85,B 0,C 180,E1 -20250,E2 -20250} C_VEL
LIN {X 0,Y 218.81,Z 388.833,A -85,B 0,C 180,E1 -20251.841,E2 -20251.841} C_VEL
LIN {X 0,Y 218.627,Z 388.665,A -85,B 0,C 180,E1 -20254.771,E2 -20254.771} C_VEL
LIN {X 0,Y 218.682,Z 387.643,A -85,B 0,C 180,E1 -20257.386,E2 -20257.386} C_VEL
LIN {X 0,Y 218.974,Z 386.467,A -85,B 0,C 180,E1 -20259.234,E2 -20259.234} C_VEL
LIN {X 0,Y 219.677,Z 383.889,A -85,B 0,C 180,E1 -20262.002,E2 -20262.002} C_VEL
LIN {X 0,Y 220.914,Z 380.33,A -85,B 0,C 180,E1 -20264.744,E2 -20264.744} C_VEL
LIN {X 0,Y 222.712,Z 375.728,A -85,B 0,C 180,E1 -20267.445,E2 -20267.445} C_VEL
LIN {X 0,Y 224.998,Z 369.953,A -85,B 0,C 180,E1 -20270.096,E2 -20270.096} C_VEL
LIN {X 0,Y 227.572,Z 362.797,A -85,B 0,C 180,E1 -20272.708,E2 -20272.708} C_VEL
LIN {X 0,Y 230.85,Z 353.926,A -85,B 0,C 180,E1 -20275.227,E2 -20275.227} C_VEL
LIN {X 0,Y 234.054,Z 344.894,A -85,B 0,C 180,E1 -20277.252,E2 -20277.252} C_VEL
LIN {X 0,Y 237.482,Z 333.803,A -85,B 0,C 180,E1 -20279.228,E2 -20279.228} C_VEL
LIN {X 0,Y 240.59,Z 322.69,A -85,B 0,C 180,E1 -20280.744,E2 -20280.744} C_VEL
LIN {X 0,Y 243.433,Z 310.417,A -85,B 0,C 180,E1 -20282.038,E2 -20282.038} C_VEL
LIN {X 0,Y 245.81,Z 297.66,A -85,B 0,C 180,E1 -20283.004,E2 -20283.004} C_VEL
LIN {X 0,Y 247.427,Z 284.398,A -85,B 0,C 180,E1 -20283.716,E2 -20283.716} C_VEL
LIN {X 0,Y 250.378,Z 238.555,A -85,B 0,C 180,E1 -20285.186,E2 -20285.186} C_VEL
LIN {X 0,Y 248.882,Z 222.435,A -85,B 0,C 180,E1 -20286.233,E2 -20286.233} C_VEL
LIN {X 0,Y 247.767,Z 214.76,A -85,B 0,C 180,E1 -20286.837,E2 -20286.837} C_VEL
LIN {X 0,Y 242.562,Z 202.741,A -85,B 0,C 180,E1 -20288.695,E2 -20288.695} C_VEL
LIN {X 0,Y 237.656,Z 193.045,A -85,B 0,C 180,E1 -20290.514,E2 -20290.514} C_VEL
LIN {X 0,Y 234.292,Z 187.175,A -85,B 0,C 180,E1 -20291.84,E2 -20291.84} C_VEL
LIN {X 0,Y 231.372,Z 182.327,A -85,B 0,C 180,E1 -20293.045,E2 -20293.045} C_VEL
LIN {X 0,Y 227.763,Z 176.57,A -85,B 0,C 180,E1 -20294.646,E2 -20294.646} C_VEL
LIN {X 0,Y 224.481,Z 171.702,A -85,B 0,C 180,E1 -20296.211,E2 -20296.211} C_VEL
LIN {X 0,Y 224.032,Z 170.663,A -85,B 0,C 180,E1 -20296.593,E2 -20296.593} C_VEL
LIN {X 0,Y 222.146,Z 164.996,A -85,B 0,C 180,E1 -20300.747,E2 -20300.747} C_VEL
LIN {X 0,Y 220.859,Z 160.967,A -85,B 0,C 180,E1 -20304.217,E2 -20304.217} C_VEL
LIN {X 0,Y 220.834,Z 160.973,A -85,B 0,C 180,E1 -20309.389,E2 -20309.389} C_VEL
LIN {X 0,Y 220.894,Z 160.959,A -85,B 0,C 180,E1 -20313.549,E2 -20313.549} C_VEL
LIN {X 0,Y 220.865,Z 160.96,A -85,B 0,C 180,E1 -20317.552,E2 -20317.552} C_VEL
LIN {X 0,Y 220.984,Z 160.953,A -85,B 0,C 180,E1 -20322.571,E2 -20322.571} C_VEL
LIN {X 0,Y 221.026,Z 160.952,A -85,B 0,C 180,E1 -20327.139,E2 -20327.139} C_VEL
LIN {X 0,Y 221.258,Z 160.925,A -85,B 0,C 180,E1 -20330.861,E2 -20330.861} C_VEL
LIN {X 0,Y 221.295,Z 160.909,A -85,B 0,C 180,E1 -20332.701,E2 -20332.701} C_VEL
LIN {X 0,Y 221.512,Z 160.894,A -85,B 0,C 180,E1 -20338.181,E2 -20338.181} C_VEL
LIN {X 0,Y 221.512,Z 160.891,A -85,B 0,C 180,E1 -20341.818,E2 -20341.818} C_VEL
LIN {X 0,Y 221.17,Z 161.051,A -85,B 0,C 180,E1 -20345.527,E2 -20345.527} C_VEL
LIN {X 0,Y 222.006,Z 163.463,A -85,B 0,C 180,E1 -20346.076,E2 -20346.076} C_VEL
LIN {X 0,Y 223.8,Z 165.527,A -85,B 0,C 180,E1 -20346.989,E2 -20346.989} C_VEL
LIN {X 0,Y 225.357,Z 166.725,A -85,B 0,C 180,E1 -20347.692,E2 -20347.692} C_VEL
LIN {X 0,Y 227.116,Z 169.785,A -85,B 0,C 180,E1 -20348.567,E2 -20348.567} C_VEL
LIN {X 0,Y 229.029,Z 171.899,A -85,B 0,C 180,E1 -20349.402,E2 -20349.402} C_VEL
LIN {X 0,Y 231.348,Z 175.362,A -85,B 0,C 180,E1 -20350.425,E2 -20350.425} C_VEL
LIN {X 0,Y 232.755,Z 177.184,A -85,B 0,C 180,E1 -20350.995,E2 -20350.995} C_VEL
LIN {X 0,Y 236.603,Z 182.753,A -85,B 0,C 180,E1 -20352.5,E2 -20352.5} C_VEL
LIN {X 0,Y 240.978,Z 189.47,A -85,B 0,C 180,E1 -20354.11,E2 -20354.11} C_VEL
LIN {X 0,Y 246.705,Z 199.174,A -85,B 0,C 180,E1 -20356.058,E2 -20356.058} C_VEL
LIN {X 0,Y 251.124,Z 207.852,A -85,B 0,C 180,E1 -20357.494,E2 -20357.494} C_VEL
LIN {X 0,Y 251.951,Z 209.689,A -85,B 0,C 180,E1 -20357.758,E2 -20357.758} C_VEL
LIN {X 0,Y 248.47,Z 264.701,A -85,B 0,C 180,E1 -20359.522,E2 -20359.522} C_VEL
LIN {X 0,Y 246.949,Z 278.208,A -85,B 0,C 180,E1 -20360.276,E2 -20360.276} C_VEL
LIN {X 0,Y 244.957,Z 291.148,A -85,B 0,C 180,E1 -20361.363,E2 -20361.363} C_VEL
LIN {X 0,Y 242.466,Z 303.287,A -85,B 0,C 180,E1 -20362.742,E2 -20362.742} C_VEL
LIN {X 0,Y 239.852,Z 313.503,A -85,B 0,C 180,E1 -20364.218,E2 -20364.218} C_VEL
LIN {X 0,Y 236.835,Z 323.89,A -85,B 0,C 180,E1 -20366.132,E2 -20366.132} C_VEL
LIN {X 0,Y 233.591,Z 333.455,A -85,B 0,C 180,E1 -20368.356,E2 -20368.356} C_VEL
LIN {X 0,Y 230.666,Z 341.161,A -85,B 0,C 180,E1 -20370.602,E2 -20370.602} C_VEL
LIN {X 0,Y 228.038,Z 347.556,A -85,B 0,C 180,E1 -20372.932,E2 -20372.932} C_VEL
LIN {X 0,Y 225.313,Z 353.732,A -85,B 0,C 180,E1 -20375.807,E2 -20375.807} C_VEL
LIN {X 0,Y 222.913,Z 358.885,A -85,B 0,C 180,E1 -20379.091,E2 -20379.091} C_VEL
LIN {X 0,Y 221.388,Z 361.926,A -85,B 0,C 180,E1 -20381.809,E2 -20381.809} C_VEL
LIN {X 0,Y 219.895,Z 364.444,A -85,B 0,C 180,E1 -20385.322,E2 -20385.322} C_VEL
LIN {X 0,Y 219.275,Z 365.24,A -85,B 0,C 180,E1 -20387.696,E2 -20387.696} C_VEL
LIN {X 0,Y 218.769,Z 365.363,A -85,B 0,C 180,E1 -20390.444,E2 -20390.444} C_VEL
LIN {X 0,Y 218.565,Z 364.453,A -85,B 0,C 180,E1 -20393.502,E2 -20393.502} C_VEL
LIN {X 0,Y 218.793,Z 362.14,A -85,B 0,C 180,E1 -20396.903,E2 -20396.903} C_VEL
LIN {X 0,Y 219.37,Z 358.901,A -85,B 0,C 180,E1 -20399.882,E2 -20399.882} C_VEL
LIN {X 0,Y 220.001,Z 355.193,A -85,B 0,C 180,E1 -20402.39,E2 -20402.39} C_VEL
LIN {X 0,Y 220.914,Z 350.155,A -85,B 0,C 180,E1 -20405.069,E2 -20405.069} C_VEL
LIN {X 0,Y 222.19,Z 343.942,A -85,B 0,C 180,E1 -20407.693,E2 -20407.693} C_VEL
LIN {X 0,Y 223.807,Z 335.866,A -85,B 0,C 180,E1 -20410.4,E2 -20410.4} C_VEL
LIN {X 0,Y 225.856,Z 325.904,A -85,B 0,C 180,E1 -20413.039,E2 -20413.039} C_VEL
LIN {X 0,Y 227.783,Z 315.271,A -85,B 0,C 180,E1 -20415.254,E2 -20415.254} C_VEL
LIN {X 0,Y 229.533,Z 304.889,A -85,B 0,C 180,E1 -20416.973,E2 -20416.973} C_VEL
LIN {X 0,Y 231.229,Z 293.269,A -85,B 0,C 180,E1 -20418.495,E2 -20418.495} C_VEL
LIN {X 0,Y 232.495,Z 281.672,A -85,B 0,C 180,E1 -20419.661,E2 -20419.661} C_VEL
LIN {X 0,Y 233.676,Z 267.637,A -85,B 0,C 180,E1 -20420.66,E2 -20420.66} C_VEL
LIN {X 0,Y 234.394,Z 254.613,A -85,B 0,C 180,E1 -20421.236,E2 -20421.236} C_VEL
LIN {X 0,Y 236.781,Z 196.692,A -85,B 0,C 180,E1 -20423.113,E2 -20423.113} C_VEL
LIN {X 0,Y 227.412,Z 174.423,A -85,B 0,C 180,E1 -20425.032,E2 -20425.032} C_VEL
LIN {X 0,Y 221.336,Z 161.692,A -85,B 0,C 180,E1 -20426.302,E2 -20426.302} C_VEL
LIN {X 0,Y 221.219,Z 160.929,A -85,B 0,C 180,E1 -20426.357,E2 -20426.357} C_VEL
LIN {X 0,Y 221.512,Z 160.893,A -85,B 0,C 180,E1 -20428.182,E2 -20428.182} C_VEL
LIN {X 0,Y 221.511,Z 160.894,A -85,B 0,C 180,E1 -20431.818,E2 -20431.818} C_VEL
LIN {X 0,Y 221.241,Z 160.929,A -85,B 0,C 180,E1 -20437.3,E2 -20437.3} C_VEL
LIN {X 0,Y 221.062,Z 160.951,A -85,B 0,C 180,E1 -20440.997,E2 -20440.997} C_VEL
LIN {X 0,Y 220.978,Z 160.959,A -85,B 0,C 180,E1 -20446.633,E2 -20446.633} C_VEL
LIN {X 0,Y 220.875,Z 160.972,A -85,B 0,C 180,E1 -20450.488,E2 -20450.488} C_VEL
LIN {X 0,Y 220.862,Z 160.972,A -85,B 0,C 180,E1 -20454.436,E2 -20454.436} C_VEL
LIN {X 0,Y 220.836,Z 160.976,A -85,B 0,C 180,E1 -20458.513,E2 -20458.513} C_VEL
LIN {X 0,Y 220.819,Z 160.979,A -85,B 0,C 180,E1 -20462.756,E2 -20462.756} C_VEL
LIN {X 0,Y 220.81,Z 160.978,A -85,B 0,C 180,E1 -20467.278,E2 -20467.278} C_VEL
LIN {X 0,Y 220.769,Z 160.976,A -85,B 0,C 180,E1 -20471.953,E2 -20471.953} C_VEL
LIN {X 0,Y 220.772,Z 160.983,A -85,B 0,C 180,E1 -20475.546,E2 -20475.546} C_VEL
LIN {X 0,Y 220.805,Z 160.969,A -85,B 0,C 180,E1 -20480.463,E2 -20480.463} C_VEL
LIN {X 0,Y 220.823,Z 160.973,A -85,B 0,C 180,E1 -20482.793,E2 -20482.793} C_VEL
LIN {X 0,Y 220.821,Z 160.975,A -85,B 0,C 180,E1 -20487.245,E2 -20487.245} C_VEL
LIN {X 0,Y 220.826,Z 160.964,A -85,B 0,C 180,E1 -20491.485,E2 -20491.485} C_VEL
LIN {X 0,Y 220.861,Z 160.973,A -85,B 0,C 180,E1 -20495.565,E2 -20495.565} C_VEL
LIN {X 0,Y 220.884,Z 160.966,A -85,B 0,C 180,E1 -20499.513,E2 -20499.513} C_VEL
LIN {X 0,Y 221.016,Z 160.942,A -85,B 0,C 180,E1 -20503.371,E2 -20503.371} C_VEL
LIN {X 0,Y 221.112,Z 160.941,A -85,B 0,C 180,E1 -20509.006,E2 -20509.006} C_VEL
LIN {X 0,Y 221.29,Z 160.909,A -85,B 0,C 180,E1 -20512.702,E2 -20512.702} C_VEL
LIN {X 0,Y 221.512,Z 160.889,A -85,B 0,C 180,E1 -20518.182,E2 -20518.182} C_VEL
LIN {X 0,Y 221.512,Z 160.884,A -85,B 0,C 180,E1 -20521.819,E2 -20521.819} C_VEL
LIN {X 0,Y 221.289,Z 160.919,A -85,B 0,C 180,E1 -20527.299,E2 -20527.299} C_VEL
LIN {X 0,Y 221.112,Z 160.936,A -85,B 0,C 180,E1 -20530.995,E2 -20530.995} C_VEL
LIN {X 0,Y 221.017,Z 160.956,A -85,B 0,C 180,E1 -20536.63,E2 -20536.63} C_VEL
LIN {X 0,Y 220.885,Z 160.965,A -85,B 0,C 180,E1 -20540.487,E2 -20540.487} C_VEL
LIN {X 0,Y 220.863,Z 160.974,A -85,B 0,C 180,E1 -20544.436,E2 -20544.436} C_VEL
LIN {X 0,Y 220.837,Z 160.978,A -85,B 0,C 180,E1 -20548.514,E2 -20548.514} C_VEL
LIN {X 0,Y 220.825,Z 160.978,A -85,B 0,C 180,E1 -20552.755,E2 -20552.755} C_VEL
LIN {X 0,Y 220.839,Z 160.975,A -85,B 0,C 180,E1 -20557.288,E2 -20557.288} C_VEL
LIN {X 0,Y 220.816,Z 160.98,A -85,B 0,C 180,E1 -20561.942,E2 -20561.942} C_VEL
LIN {X 0,Y 220.816,Z 160.978,A -85,B 0,C 180,E1 -20562.506,E2 -20562.506} C_VEL
LIN {X 0,Y 220.148,Z 161.063,A -85,B 0,C 180,E1 -20563.516,E2 -20563.516} C_VEL
LIN {X 0,Y 217.29,Z 161.416,A -85,B 0,C 180,E1 -20565.102,E2 -20565.102} C_VEL
LIN {X 0,Y 214.392,Z 161.779,A -85,B 0,C 180,E1 -20566.727,E2 -20566.727} C_VEL
LIN {X 0,Y 213.706,Z 161.859,A -85,B 0,C 180,E1 -20567.784,E2 -20567.784} C_VEL
LIN {X 0,Y 213.777,Z 161.936,A -85,B 0,C 180,E1 -20569.823,E2 -20569.823} C_VEL
LIN {X 0,Y 215.936,Z 170.946,A -85,B 0,C 180,E1 -20573.734,E2 -20573.734} C_VEL
LIN {X 0,Y 217.029,Z 176.215,A -85,B 0,C 180,E1 -20575.836,E2 -20575.836} C_VEL
LIN {X 0,Y 224.516,Z 196.119,A -85,B 0,C 180,E1 -20577.587,E2 -20577.587} C_VEL
LIN {X 0,Y 228.449,Z 229.227,A -85,B 0,C 180,E1 -20579.326,E2 -20579.326} C_VEL
LIN {X 0,Y 228.991,Z 235.613,A -85,B 0,C 180,E1 -20579.627,E2 -20579.627} C_VEL
LIN {X 0,Y 226.858,Z 285.91,A -85,B 0,C 180,E1 -20581.366,E2 -20581.366} C_VEL
LIN {X 0,Y 225.745,Z 298.461,A -85,B 0,C 180,E1 -20582.098,E2 -20582.098} C_VEL
LIN {X 0,Y 224.314,Z 310.376,A -85,B 0,C 180,E1 -20583.106,E2 -20583.106} C_VEL
LIN {X 0,Y 222.412,Z 322.562,A -85,B 0,C 180,E1 -20584.498,E2 -20584.498} C_VEL
LIN {X 0,Y 220.578,Z 332.869,A -85,B 0,C 180,E1 -20586.031,E2 -20586.031} C_VEL
LIN {X 0,Y 218.409,Z 343.561,A -85,B 0,C 180,E1 -20588.033,E2 -20588.033} C_VEL
LIN {X 0,Y 216.549,Z 352.984,A -85,B 0,C 180,E1 -20590.252,E2 -20590.252} C_VEL
LIN {X 0,Y 215.108,Z 360.426,A -85,B 0,C 180,E1 -20592.409,E2 -20592.409} C_VEL
LIN {X 0,Y 213.577,Z 368.293,A -85,B 0,C 180,E1 -20595.225,E2 -20595.225} C_VEL
LIN {X 0,Y 212.58,Z 373.639,A -85,B 0,C 180,E1 -20597.591,E2 -20597.591} C_VEL
LIN {X 0,Y 211.992,Z 378.81,A -85,B 0,C 180,E1 -20600.459,E2 -20600.459} C_VEL
LIN {X 0,Y 211.719,Z 382.779,A -85,B 0,C 180,E1 -20603.328,E2 -20603.328} C_VEL
LIN {X 0,Y 211.723,Z 385.661,A -85,B 0,C 180,E1 -20606.193,E2 -20606.193} C_VEL
LIN {X 0,Y 211.786,Z 386.991,A -85,B 0,C 180,E1 -20608.098,E2 -20608.098} C_VEL
LIN {X 0,Y 211.824,Z 387.902,A -85,B 0,C 180,E1 -20610,E2 -20610} C_VEL
LIN {X 0,Y 211.736,Z 388.395,A -85,B 0,C 180,E1 -20611.902,E2 -20611.902} C_VEL
LIN {X 0,Y 211.546,Z 388.329,A -85,B 0,C 180,E1 -20614.678,E2 -20614.678} C_VEL
LIN {X 0,Y 211.62,Z 387.339,A -85,B 0,C 180,E1 -20617.634,E2 -20617.634} C_VEL
LIN {X 0,Y 211.921,Z 386.204,A -85,B 0,C 180,E1 -20619.545,E2 -20619.545} C_VEL
LIN {X 0,Y 212.385,Z 384.658,A -85,B 0,C 180,E1 -20621.452,E2 -20621.452} C_VEL
LIN {X 0,Y 213.501,Z 381.537,A -85,B 0,C 180,E1 -20624.293,E2 -20624.293} C_VEL
LIN {X 0,Y 215.282,Z 377.392,A -85,B 0,C 180,E1 -20627.086,E2 -20627.086} C_VEL
LIN {X 0,Y 217.474,Z 372.122,A -85,B 0,C 180,E1 -20629.835,E2 -20629.835} C_VEL
LIN {X 0,Y 220.072,Z 365.557,A -85,B 0,C 180,E1 -20632.533,E2 -20632.533} C_VEL
LIN {X 0,Y 223.248,Z 357.444,A -85,B 0,C 180,E1 -20635.15,E2 -20635.15} C_VEL
LIN {X 0,Y 227.1,Z 347.465,A -85,B 0,C 180,E1 -20637.658,E2 -20637.658} C_VEL
LIN {X 0,Y 230.598,Z 337.091,A -85,B 0,C 180,E1 -20639.686,E2 -20639.686} C_VEL
LIN {X 0,Y 234.149,Z 325.503,A -85,B 0,C 180,E1 -20641.433,E2 -20641.433} C_VEL
LIN {X 0,Y 237.071,Z 314.132,A -85,B 0,C 180,E1 -20642.753,E2 -20642.753} C_VEL
LIN {X 0,Y 239.764,Z 301.302,A -85,B 0,C 180,E1 -20643.844,E2 -20643.844} C_VEL
LIN {X 0,Y 241.763,Z 288.079,A -85,B 0,C 180,E1 -20644.648,E2 -20644.648} C_VEL
LIN {X 0,Y 242.991,Z 273.369,A -85,B 0,C 180,E1 -20645.218,E2 -20645.218} C_VEL
LIN {X 0,Y 245.146,Z 238.402,A -85,B 0,C 180,E1 -20646.341,E2 -20646.341} C_VEL
LIN {X 0,Y 243.27,Z 219.062,A -85,B 0,C 180,E1 -20647.711,E2 -20647.711} C_VEL
LIN {X 0,Y 239.901,Z 210.535,A -85,B 0,C 180,E1 -20648.995,E2 -20648.995} C_VEL
LIN {X 0,Y 234.42,Z 198.904,A -85,B 0,C 180,E1 -20651.151,E2 -20651.151} C_VEL
LIN {X 0,Y 229.863,Z 190.821,A -85,B 0,C 180,E1 -20653.041,E2 -20653.041} C_VEL
LIN {X 0,Y 227.855,Z 187.476,A -85,B 0,C 180,E1 -20653.929,E2 -20653.929} C_VEL
LIN {X 0,Y 224.582,Z 182.088,A -85,B 0,C 180,E1 -20655.478,E2 -20655.478} C_VEL
LIN {X 0,Y 221.299,Z 176.904,A -85,B 0,C 180,E1 -20657.141,E2 -20657.141} C_VEL
LIN {X 0,Y 217.206,Z 171.253,A -85,B 0,C 180,E1 -20659.423,E2 -20659.423} C_VEL
LIN {X 0,Y 216.567,Z 170,A -85,B 0,C 180,E1 -20659.835,E2 -20659.835} C_VEL
LIN {X 0,Y 214.999,Z 165.205,A -85,B 0,C 180,E1 -20663.956,E2 -20663.956} C_VEL
LIN {X 0,Y 213.79,Z 161.847,A -85,B 0,C 180,E1 -20667.571,E2 -20667.571} C_VEL
LIN {X 0,Y 213.826,Z 161.845,A -85,B 0,C 180,E1 -20672.603,E2 -20672.603} C_VEL
LIN {X 0,Y 213.819,Z 161.838,A -85,B 0,C 180,E1 -20676.973,E2 -20676.973} C_VEL
LIN {X 0,Y 213.962,Z 161.83,A -85,B 0,C 180,E1 -20682.805,E2 -20682.805} C_VEL
LIN {X 0,Y 213.98,Z 161.83,A -85,B 0,C 180,E1 -20686.708,E2 -20686.708} C_VEL
LIN {X 0,Y 214.197,Z 161.805,A -85,B 0,C 180,E1 -20690.557,E2 -20690.557} C_VEL
LIN {X 0,Y 214.111,Z 161.815,A -85,B 0,C 180,E1 -20694.348,E2 -20694.348} C_VEL
LIN {X 0,Y 214.445,Z 161.774,A -85,B 0,C 180,E1 -20698.122,E2 -20698.122} C_VEL
LIN {X 0,Y 214.55,Z 161.751,A -85,B 0,C 180,E1 -20700,E2 -20700} C_VEL
LIN {X 0,Y 214.385,Z 161.917,A -85,B 0,C 180,E1 -20702.231,E2 -20702.231} C_VEL
LIN {X 0,Y 215.153,Z 164.421,A -85,B 0,C 180,E1 -20702.867,E2 -20702.867} C_VEL
LIN {X 0,Y 216.861,Z 166.565,A -85,B 0,C 180,E1 -20703.931,E2 -20703.931} C_VEL
LIN {X 0,Y 218.575,Z 167.843,A -85,B 0,C 180,E1 -20704.853,E2 -20704.853} C_VEL
LIN {X 0,Y 220.46,Z 170.946,A -85,B 0,C 180,E1 -20705.946,E2 -20705.946} C_VEL
LIN {X 0,Y 222.617,Z 173.011,A -85,B 0,C 180,E1 -20707.026,E2 -20707.026} C_VEL
LIN {X 0,Y 225.086,Z 176.641,A -85,B 0,C 180,E1 -20708.246,E2 -20708.246} C_VEL
LIN {X 0,Y 226.305,Z 178.248,A -85,B 0,C 180,E1 -20708.81,E2 -20708.81} C_VEL
LIN {X 0,Y 229.888,Z 183.393,A -85,B 0,C 180,E1 -20710.414,E2 -20710.414} C_VEL
LIN {X 0,Y 233.155,Z 188.15,A -85,B 0,C 180,E1 -20711.748,E2 -20711.748} C_VEL
LIN {X 0,Y 237.349,Z 194.753,A -85,B 0,C 180,E1 -20713.375,E2 -20713.375} C_VEL
LIN {X 0,Y 242.726,Z 204.124,A -85,B 0,C 180,E1 -20715.306,E2 -20715.306} C_VEL
LIN {X 0,Y 246.715,Z 212.207,A -85,B 0,C 180,E1 -20716.683,E2 -20716.683} C_VEL
LIN {X 0,Y 243.23,Z 264.989,A -85,B 0,C 180,E1 -20718.415,E2 -20718.415} C_VEL
LIN {X 0,Y 241.674,Z 278.188,A -85,B 0,C 180,E1 -20719.151,E2 -20719.151} C_VEL
LIN {X 0,Y 239.653,Z 290.908,A -85,B 0,C 180,E1 -20720.213,E2 -20720.213} C_VEL
LIN {X 0,Y 237.116,Z 302.904,A -85,B 0,C 180,E1 -20721.576,E2 -20721.576} C_VEL
LIN {X 0,Y 234.002,Z 314.637,A -85,B 0,C 180,E1 -20723.296,E2 -20723.296} C_VEL
LIN {X 0,Y 230.834,Z 324.801,A -85,B 0,C 180,E1 -20725.229,E2 -20725.229} C_VEL
LIN {X 0,Y 227.235,Z 334.784,A -85,B 0,C 180,E1 -20727.64,E2 -20727.64} C_VEL
LIN {X 0,Y 223.961,Z 342.864,A -85,B 0,C 180,E1 -20730.138,E2 -20730.138} C_VEL
LIN {X 0,Y 221.006,Z 349.455,A -85,B 0,C 180,E1 -20732.724,E2 -20732.724} C_VEL
LIN {X 0,Y 218.489,Z 354.748,A -85,B 0,C 180,E1 -20735.379,E2 -20735.379} C_VEL
LIN {X 0,Y 216.038,Z 359.645,A -85,B 0,C 180,E1 -20738.671,E2 -20738.671} C_VEL
LIN {X 0,Y 214.633,Z 362.28,A -85,B 0,C 180,E1 -20741.139,E2 -20741.139} C_VEL
LIN {X 0,Y 213.406,Z 364.259,A -85,B 0,C 180,E1 -20743.755,E2 -20743.755} C_VEL
LIN {X 0,Y 212.38,Z 365.53,A -85,B 0,C 180,E1 -20746.72,E2 -20746.72} C_VEL
LIN {X 0,Y 211.78,Z 365.814,A -85,B 0,C 180,E1 -20749.752,E2 -20749.752} C_VEL
LIN {X 0,Y 211.505,Z 364.866,A -85,B 0,C 180,E1 -20753.265,E2 -20753.265} C_VEL
LIN {X 0,Y 211.61,Z 363.088,A -85,B 0,C 180,E1 -20756.129,E2 -20756.129} C_VEL
LIN {X 0,Y 212.165,Z 359.802,A -85,B 0,C 180,E1 -20759.457,E2 -20759.457} C_VEL
LIN {X 0,Y 212.936,Z 355.584,A -85,B 0,C 180,E1 -20762.479,E2 -20762.479} C_VEL
LIN {X 0,Y 214.065,Z 349.588,A -85,B 0,C 180,E1 -20765.704,E2 -20765.704} C_VEL
LIN {X 0,Y 215.464,Z 342.945,A -85,B 0,C 180,E1 -20768.473,E2 -20768.473} C_VEL
LIN {X 0,Y 217.148,Z 335.016,A -85,B 0,C 180,E1 -20771.116,E2 -20771.116} C_VEL
LIN {X 0,Y 219.135,Z 325.469,A -85,B 0,C 180,E1 -20773.66,E2 -20773.66} C_VEL
LIN {X 0,Y 221.195,Z 314.388,A -85,B 0,C 180,E1 -20775.98,E2 -20775.98} C_VEL
LIN {X 0,Y 223.146,Z 302.99,A -85,B 0,C 180,E1 -20777.855,E2 -20777.855} C_VEL
LIN {X 0,Y 224.913,Z 290.54,A -85,B 0,C 180,E1 -20779.422,E2 -20779.422} C_VEL
LIN {X 0,Y 226.236,Z 278.001,A -85,B 0,C 180,E1 -20780.614,E2 -20780.614} C_VEL
LIN {X 0,Y 227.326,Z 264.654,A -85,B 0,C 180,E1 -20781.476,E2 -20781.476} C_VEL
LIN {X 0,Y 228.198,Z 247.047,A -85,B 0,C 180,E1 -20782.148,E2 -20782.148} C_VEL
LIN {X 0,Y 230.253,Z 198.231,A -85,B 0,C 180,E1 -20783.776,E2 -20783.776} C_VEL
LIN {X 0,Y 221.081,Z 176.63,A -85,B 0,C 180,E1 -20785.734,E2 -20785.734} C_VEL
LIN {X 0,Y 214.481,Z 162.764,A -85,B 0,C 180,E1 -20787.182,E2 -20787.182} C_VEL
LIN {X 0,Y 214.291,Z 161.793,A -85,B 0,C 180,E1 -20787.297,E2 -20787.297} C_VEL
LIN {X 0,Y 214.55,Z 161.76,A -85,B 0,C 180,E1 -20790,E2 -20790} C_VEL
LIN {X 0,Y 214.444,Z 161.775,A -85,B 0,C 180,E1 -20791.878,E2 -20791.878} C_VEL
LIN {X 0,Y 214.182,Z 161.807,A -85,B 0,C 180,E1 -20797.542,E2 -20797.542} C_VEL
LIN {X 0,Y 213.993,Z 161.831,A -85,B 0,C 180,E1 -20801.365,E2 -20801.365} C_VEL
LIN {X 0,Y 213.902,Z 161.84,A -85,B 0,C 180,E1 -20805.239,E2 -20805.239} C_VEL
LIN {X 0,Y 213.813,Z 161.851,A -85,B 0,C 180,E1 -20809.19,E2 -20809.19} C_VEL
LIN {X 0,Y 213.81,Z 161.85,A -85,B 0,C 180,E1 -20813.231,E2 -20813.231} C_VEL
LIN {X 0,Y 213.829,Z 161.846,A -85,B 0,C 180,E1 -20817.45,E2 -20817.45} C_VEL
LIN {X 0,Y 213.777,Z 161.853,A -85,B 0,C 180,E1 -20821.736,E2 -20821.736} C_VEL
LIN {X 0,Y 213.744,Z 161.86,A -85,B 0,C 180,E1 -20826.288,E2 -20826.288} C_VEL
LIN {X 0,Y 213.711,Z 161.853,A -85,B 0,C 180,E1 -20831.125,E2 -20831.125} C_VEL
LIN {X 0,Y 213.705,Z 161.861,A -85,B 0,C 180,E1 -20833.679,E2 -20833.679} C_VEL
LIN {X 0,Y 213.705,Z 161.864,A -85,B 0,C 180,E1 -20836.344,E2 -20836.344} C_VEL
LIN {X 0,Y 213.733,Z 161.85,A -85,B 0,C 180,E1 -20841.336,E2 -20841.336} C_VEL
LIN {X 0,Y 213.767,Z 161.857,A -85,B 0,C 180,E1 -20846.02,E2 -20846.02} C_VEL
LIN {X 0,Y 213.759,Z 161.842,A -85,B 0,C 180,E1 -20850.451,E2 -20850.451} C_VEL
LIN {X 0,Y 213.797,Z 161.85,A -85,B 0,C 180,E1 -20854.702,E2 -20854.702} C_VEL
LIN {X 0,Y 213.803,Z 161.849,A -85,B 0,C 180,E1 -20858.803,E2 -20858.803} C_VEL
LIN {X 0,Y 213.943,Z 161.82,A -85,B 0,C 180,E1 -20862.804,E2 -20862.804} C_VEL
LIN {X 0,Y 213.98,Z 161.828,A -85,B 0,C 180,E1 -20866.709,E2 -20866.709} C_VEL
LIN {X 0,Y 214.168,Z 161.802,A -85,B 0,C 180,E1 -20870.557,E2 -20870.557} C_VEL
LIN {X 0,Y 214.228,Z 161.788,A -85,B 0,C 180,E1 -20872.46,E2 -20872.46} C_VEL
LIN {X 0,Y 214.446,Z 161.769,A -85,B 0,C 180,E1 -20878.122,E2 -20878.122} C_VEL
LIN {X 0,Y 214.55,Z 161.755,A -85,B 0,C 180,E1 -20880,E2 -20880} C_VEL
LIN {X 0,Y 214.445,Z 161.763,A -85,B 0,C 180,E1 -20881.878,E2 -20881.878} C_VEL
LIN {X 0,Y 214.227,Z 161.798,A -85,B 0,C 180,E1 -20887.541,E2 -20887.541} C_VEL
LIN {X 0,Y 214.045,Z 161.814,A -85,B 0,C 180,E1 -20891.362,E2 -20891.362} C_VEL
LIN {X 0,Y 213.934,Z 161.835,A -85,B 0,C 180,E1 -20895.237,E2 -20895.237} C_VEL
LIN {X 0,Y 213.836,Z 161.843,A -85,B 0,C 180,E1 -20899.188,E2 -20899.188} C_VEL
LIN {X 0,Y 213.811,Z 161.851,A -85,B 0,C 180,E1 -20903.232,E2 -20903.232} C_VEL
LIN {X 0,Y 213.83,Z 161.846,A -85,B 0,C 180,E1 -20907.45,E2 -20907.45} C_VEL
LIN {X 0,Y 213.78,Z 161.854,A -85,B 0,C 180,E1 -20911.736,E2 -20911.736} C_VEL
LIN {X 0,Y 213.755,Z 161.861,A -85,B 0,C 180,E1 -20916.287,E2 -20916.287} C_VEL
LIN {X 0,Y 213.741,Z 161.86,A -85,B 0,C 180,E1 -20921.119,E2 -20921.119} C_VEL
LIN {X 0,Y 213.776,Z 161.856,A -85,B 0,C 180,E1 -20923.676,E2 -20923.676} C_VEL
LIN {X 0,Y 213.706,Z 161.859,A -85,B 0,C 180,E1 -20927.784,E2 -20927.784} C_VEL
LIN {X 0,Y 213.137,Z 162.423,A -85,B 0,C 180,E1 -20928.823,E2 -20928.823} C_VEL
LIN {X 0,Y 211.861,Z 163.81,A -85,B 0,C 180,E1 -20929.784,E2 -20929.784} C_VEL
LIN {X 0,Y 209.118,Z 167.949,A -85,B 0,C 180,E1 -20931.584,E2 -20931.584} C_VEL
LIN {X 0,Y 208.625,Z 170.622,A -85,B 0,C 180,E1 -20932.667,E2 -20932.667} C_VEL
LIN {X 0,Y 208.689,Z 170.986,A -85,B 0,C 180,E1 -20932.825,E2 -20932.825} C_VEL
LIN {X 0,Y 209.711,Z 175.748,A -85,B 0,C 180,E1 -20934.822,E2 -20934.822} C_VEL
LIN {X 0,Y 218.281,Z 198.346,A -85,B 0,C 180,E1 -20936.907,E2 -20936.907} C_VEL
LIN {X 0,Y 222.145,Z 231.991,A -85,B 0,C 180,E1 -20938.726,E2 -20938.726} C_VEL
LIN {X 0,Y 222.388,Z 237.58,A -85,B 0,C 180,E1 -20938.975,E2 -20938.975} C_VEL
LIN {X 0,Y 220.279,Z 285.652,A -85,B 0,C 180,E1 -20940.69,E2 -20940.69} C_VEL
LIN {X 0,Y 219.128,Z 298.156,A -85,B 0,C 180,E1 -20941.44,E2 -20941.44} C_VEL
LIN {X 0,Y 217.661,Z 310.051,A -85,B 0,C 180,E1 -20942.475,E2 -20942.475} C_VEL
LIN {X 0,Y 215.697,Z 322.219,A -85,B 0,C 180,E1 -20943.905,E2 -20943.905} C_VEL
LIN {X 0,Y 213.447,Z 333.793,A -85,B 0,C 180,E1 -20945.696,E2 -20945.696} C_VEL
LIN {X 0,Y 211.384,Z 344.297,A -85,B 0,C 180,E1 -20947.778,E2 -20947.778} C_VEL
LIN {X 0,Y 209.616,Z 352.706,A -85,B 0,C 180,E1 -20949.849,E2 -20949.849} C_VEL
LIN {X 0,Y 207.973,Z 360.795,A -85,B 0,C 180,E1 -20952.294,E2 -20952.294} C_VEL
LIN {X 0,Y 206.433,Z 368.493,A -85,B 0,C 180,E1 -20955.206,E2 -20955.206} C_VEL
LIN {X 0,Y 205.335,Z 374.657,A -85,B 0,C 180,E1 -20958.149,E2 -20958.149} C_VEL
LIN {X 0,Y 204.823,Z 379.522,A -85,B 0,C 180,E1 -20961.118,E2 -20961.118} C_VEL
LIN {X 0,Y 204.651,Z 383.208,A -85,B 0,C 180,E1 -20964.087,E2 -20964.087} C_VEL
LIN {X 0,Y 204.648,Z 385.083,A -85,B 0,C 180,E1 -20966.062,E2 -20966.062} C_VEL
LIN {X 0,Y 204.717,Z 386.467,A -85,B 0,C 180,E1 -20968.033,E2 -20968.033} C_VEL
LIN {X 0,Y 204.754,Z 387.415,A -85,B 0,C 180,E1 -20970,E2 -20970} C_VEL
LIN {X 0,Y 204.662,Z 387.946,A -85,B 0,C 180,E1 -20971.968,E2 -20971.968} C_VEL
LIN {X 0,Y 204.468,Z 387.988,A -85,B 0,C 180,E1 -20974.586,E2 -20974.586} C_VEL
LIN {X 0,Y 204.556,Z 387.044,A -85,B 0,C 180,E1 -20977.899,E2 -20977.899} C_VEL
LIN {X 0,Y 205.396,Z 384.471,A -85,B 0,C 180,E1 -20981.847,E2 -20981.847} C_VEL
LIN {X 0,Y 206.599,Z 381.42,A -85,B 0,C 180,E1 -20984.781,E2 -20984.781} C_VEL
LIN {X 0,Y 208.471,Z 377.362,A -85,B 0,C 180,E1 -20987.662,E2 -20987.662} C_VEL
LIN {X 0,Y 211.255,Z 371.221,A -85,B 0,C 180,E1 -20990.954,E2 -20990.954} C_VEL
LIN {X 0,Y 214.016,Z 364.578,A -85,B 0,C 180,E1 -20993.72,E2 -20993.72} C_VEL
LIN {X 0,Y 217.498,Z 356.387,A -85,B 0,C 180,E1 -20996.378,E2 -20996.378} C_VEL
LIN {X 0,Y 220.873,Z 348.077,A -85,B 0,C 180,E1 -20998.508,E2 -20998.508} C_VEL
LIN {X 0,Y 224.505,Z 338.002,A -85,B 0,C 180,E1 -21000.577,E2 -21000.577} C_VEL
LIN {X 0,Y 228.176,Z 326.686,A -85,B 0,C 180,E1 -21002.355,E2 -21002.355} C_VEL
LIN {X 0,Y 231.2,Z 315.717,A -85,B 0,C 180,E1 -21003.694,E2 -21003.694} C_VEL
LIN {X 0,Y 233.983,Z 303.702,A -85,B 0,C 180,E1 -21004.798,E2 -21004.798} C_VEL
LIN {X 0,Y 236.215,Z 290.643,A -85,B 0,C 180,E1 -21005.659,E2 -21005.659} C_VEL
LIN {X 0,Y 237.624,Z 277.11,A -85,B 0,C 180,E1 -21006.265,E2 -21006.265} C_VEL
LIN {X 0,Y 240.105,Z 239.647,A -85,B 0,C 180,E1 -21007.49,E2 -21007.49} C_VEL
LIN {X 0,Y 238.514,Z 221.911,A -85,B 0,C 180,E1 -21008.781,E2 -21008.781} C_VEL
LIN {X 0,Y 234.103,Z 211.197,A -85,B 0,C 180,E1 -21010.565,E2 -21010.565} C_VEL
LIN {X 0,Y 230.087,Z 202.763,A -85,B 0,C 180,E1 -21012.274,E2 -21012.274} C_VEL
LIN {X 0,Y 226.703,Z 196.517,A -85,B 0,C 180,E1 -21013.776,E2 -21013.776} C_VEL
LIN {X 0,Y 224.343,Z 192.438,A -85,B 0,C 180,E1 -21014.894,E2 -21014.894} C_VEL
LIN {X 0,Y 221.614,Z 187.822,A -85,B 0,C 180,E1 -21016.253,E2 -21016.253} C_VEL
LIN {X 0,Y 217.859,Z 181.883,A -85,B 0,C 180,E1 -21018.295,E2 -21018.295} C_VEL
LIN {X 0,Y 214.345,Z 176.612,A -85,B 0,C 180,E1 -21020.407,E2 -21020.407} C_VEL
LIN {X 0,Y 209.604,Z 170.11,A -85,B 0,C 180,E1 -21023.734,E2 -21023.734} C_VEL
LIN {X 0,Y 208.892,Z 168.701,A -85,B 0,C 180,E1 -21024.462,E2 -21024.462} C_VEL
LIN {X 0,Y 207.869,Z 165.751,A -85,B 0,C 180,E1 -21027.697,E2 -21027.697} C_VEL
LIN {X 0,Y 206.764,Z 162.729,A -85,B 0,C 180,E1 -21032.097,E2 -21032.097} C_VEL
LIN {X 0,Y 206.754,Z 162.72,A -85,B 0,C 180,E1 -21036.603,E2 -21036.603} C_VEL
LIN {X 0,Y 206.873,Z 162.706,A -85,B 0,C 180,E1 -21042.196,E2 -21042.196} C_VEL
LIN {X 0,Y 206.913,Z 162.705,A -85,B 0,C 180,E1 -21046.245,E2 -21046.245} C_VEL
LIN {X 0,Y 207.133,Z 162.681,A -85,B 0,C 180,E1 -21050.232,E2 -21050.232} C_VEL
LIN {X 0,Y 207.074,Z 162.69,A -85,B 0,C 180,E1 -21054.156,E2 -21054.156} C_VEL
LIN {X 0,Y 207.37,Z 162.811,A -85,B 0,C 180,E1 -21057.814,E2 -21057.814} C_VEL
LIN {X 0,Y 208.308,Z 165.306,A -85,B 0,C 180,E1 -21058.791,E2 -21058.791} C_VEL
LIN {X 0,Y 210.673,Z 167.71,A -85,B 0,C 180,E1 -21060.599,E2 -21060.599} C_VEL
LIN {X 0,Y 211.99,Z 168.618,A -85,B 0,C 180,E1 -21061.475,E2 -21061.475} C_VEL
LIN {X 0,Y 213.475,Z 171.647,A -85,B 0,C 180,E1 -21062.594,E2 -21062.594} C_VEL
LIN {X 0,Y 216.206,Z 174.328,A -85,B 0,C 180,E1 -21064.231,E2 -21064.231} C_VEL
LIN {X 0,Y 218.443,Z 177.615,A -85,B 0,C 180,E1 -21065.538,E2 -21065.538} C_VEL
LIN {X 0,Y 220.062,Z 179.336,A -85,B 0,C 180,E1 -21066.389,E2 -21066.389} C_VEL
LIN {X 0,Y 223.837,Z 184.829,A -85,B 0,C 180,E1 -21068.307,E2 -21068.307} C_VEL
LIN {X 0,Y 228.833,Z 192.001,A -85,B 0,C 180,E1 -21070.578,E2 -21070.578} C_VEL
LIN {X 0,Y 235.141,Z 202.291,A -85,B 0,C 180,E1 -21073.141,E2 -21073.141} C_VEL
LIN {X 0,Y 240.646,Z 212.591,A -85,B 0,C 180,E1 -21075.196,E2 -21075.196} C_VEL
LIN {X 0,Y 241.62,Z 214.735,A -85,B 0,C 180,E1 -21075.553,E2 -21075.553} C_VEL
LIN {X 0,Y 238.165,Z 265.025,A -85,B 0,C 180,E1 -21077.229,E2 -21077.229} C_VEL
LIN {X 0,Y 236.513,Z 278.4,A -85,B 0,C 180,E1 -21077.978,E2 -21077.978} C_VEL
LIN {X 0,Y 234.438,Z 290.975,A -85,B 0,C 180,E1 -21079.04,E2 -21079.04} C_VEL
LIN {X 0,Y 231.788,Z 302.886,A -85,B 0,C 180,E1 -21080.402,E2 -21080.402} C_VEL
LIN {X 0,Y 228.439,Z 314.932,A -85,B 0,C 180,E1 -21082.184,E2 -21082.184} C_VEL
LIN {X 0,Y 225.232,Z 324.888,A -85,B 0,C 180,E1 -21084.102,E2 -21084.102} C_VEL
LIN {X 0,Y 221.74,Z 334.15,A -85,B 0,C 180,E1 -21086.342,E2 -21086.342} C_VEL
LIN {X 0,Y 218.134,Z 342.538,A -85,B 0,C 180,E1 -21088.899,E2 -21088.899} C_VEL
LIN {X 0,Y 214.806,Z 349.647,A -85,B 0,C 180,E1 -21091.717,E2 -21091.717} C_VEL
LIN {X 0,Y 212.301,Z 354.643,A -85,B 0,C 180,E1 -21094.247,E2 -21094.247} C_VEL
LIN {X 0,Y 210.013,Z 358.916,A -85,B 0,C 180,E1 -21097.039,E2 -21097.039} C_VEL
LIN {X 0,Y 208.203,Z 362.164,A -85,B 0,C 180,E1 -21099.893,E2 -21099.893} C_VEL
LIN {X 0,Y 206.681,Z 364.484,A -85,B 0,C 180,E1 -21102.849,E2 -21102.849} C_VEL
LIN {X 0,Y 205.261,Z 366.046,A -85,B 0,C 180,E1 -21106.782,E2 -21106.782} C_VEL
LIN {X 0,Y 204.775,Z 366.229,A -85,B 0,C 180,E1 -21109.301,E2 -21109.301} C_VEL
LIN {X 0,Y 204.414,Z 365.604,A -85,B 0,C 180,E1 -21112.257,E2 -21112.257} C_VEL
LIN {X 0,Y 204.48,Z 363.809,A -85,B 0,C 180,E1 -21115.576,E2 -21115.576} C_VEL
LIN {X 0,Y 204.974,Z 360.639,A -85,B 0,C 180,E1 -21119.049,E2 -21119.049} C_VEL
LIN {X 0,Y 205.856,Z 355.963,A -85,B 0,C 180,E1 -21122.579,E2 -21122.579} C_VEL
LIN {X 0,Y 206.789,Z 351.005,A -85,B 0,C 180,E1 -21125.397,E2 -21125.397} C_VEL
LIN {X 0,Y 208.164,Z 344.794,A -85,B 0,C 180,E1 -21128.199,E2 -21128.199} C_VEL
LIN {X 0,Y 209.785,Z 337.201,A -85,B 0,C 180,E1 -21130.936,E2 -21130.936} C_VEL
LIN {X 0,Y 211.616,Z 328.971,A -85,B 0,C 180,E1 -21133.322,E2 -21133.322} C_VEL
LIN {X 0,Y 213.643,Z 318.748,A -85,B 0,C 180,E1 -21135.717,E2 -21135.717} C_VEL
LIN {X 0,Y 215.723,Z 307.526,A -85,B 0,C 180,E1 -21137.785,E2 -21137.785} C_VEL
LIN {X 0,Y 217.669,Z 295.235,A -85,B 0,C 180,E1 -21139.536,E2 -21139.536} C_VEL
LIN {X 0,Y 219.209,Z 282.545,A -85,B 0,C 180,E1 -21140.908,E2 -21140.908} C_VEL
LIN {X 0,Y 220.486,Z 268.657,A -85,B 0,C 180,E1 -21141.953,E2 -21141.953} C_VEL
LIN {X 0,Y 221.297,Z 254.98,A -85,B 0,C 180,E1 -21142.591,E2 -21142.591} C_VEL
LIN {X 0,Y 223.691,Z 199.904,A -85,B 0,C 180,E1 -21144.481,E2 -21144.481} C_VEL
LIN {X 0,Y 215.315,Z 180.084,A -85,B 0,C 180,E1 -21146.341,E2 -21146.341} C_VEL
LIN {X 0,Y 207.592,Z 163.611,A -85,B 0,C 180,E1 -21148.121,E2 -21148.121} C_VEL
LIN {X 0,Y 207.42,Z 162.648,A -85,B 0,C 180,E1 -21148.24,E2 -21148.24} C_VEL
LIN {X 0,Y 207.515,Z 162.636,A -85,B 0,C 180,E1 -21150,E2 -21150} C_VEL
LIN {X 0,Y 207.38,Z 162.654,A -85,B 0,C 180,E1 -21151.942,E2 -21151.942} C_VEL
LIN {X 0,Y 207.127,Z 162.685,A -85,B 0,C 180,E1 -21157.801,E2 -21157.801} C_VEL
LIN {X 0,Y 206.916,Z 162.711,A -85,B 0,C 180,E1 -21161.759,E2 -21161.759} C_VEL
LIN {X 0,Y 206.83,Z 162.72,A -85,B 0,C 180,E1 -21165.774,E2 -21165.774} C_VEL
LIN {X 0,Y 206.748,Z 162.73,A -85,B 0,C 180,E1 -21169.873,E2 -21169.873} C_VEL
LIN {X 0,Y 206.747,Z 162.729,A -85,B 0,C 180,E1 -21174.074,E2 -21174.074} C_VEL
LIN {X 0,Y 206.744,Z 162.731,A -85,B 0,C 180,E1 -21178.419,E2 -21178.419} C_VEL
LIN {X 0,Y 206.703,Z 162.737,A -85,B 0,C 180,E1 -21182.957,E2 -21182.957} C_VEL
LIN {X 0,Y 206.679,Z 162.739,A -85,B 0,C 180,E1 -21187.74,E2 -21187.74} C_VEL
LIN {X 0,Y 206.641,Z 162.733,A -85,B 0,C 180,E1 -21191.563,E2 -21191.563} C_VEL
LIN {X 0,Y 206.632,Z 162.745,A -85,B 0,C 180,E1 -21195.582,E2 -21195.582} C_VEL
LIN {X 0,Y 206.662,Z 162.731,A -85,B 0,C 180,E1 -21199.75,E2 -21199.75} C_VEL
LIN {X 0,Y 206.731,Z 162.731,A -85,B 0,C 180,E1 -21204.695,E2 -21204.695} C_VEL
LIN {X 0,Y 206.707,Z 162.727,A -85,B 0,C 180,E1 -21209.337,E2 -21209.337} C_VEL
LIN {X 0,Y 206.73,Z 162.729,A -85,B 0,C 180,E1 -21213.772,E2 -21213.772} C_VEL
LIN {X 0,Y 206.738,Z 162.73,A -85,B 0,C 180,E1 -21218.042,E2 -21218.042} C_VEL
LIN {X 0,Y 206.872,Z 162.699,A -85,B 0,C 180,E1 -21222.197,E2 -21222.197} C_VEL
LIN {X 0,Y 206.913,Z 162.708,A -85,B 0,C 180,E1 -21226.246,E2 -21226.246} C_VEL
LIN {X 0,Y 207.106,Z 162.681,A -85,B 0,C 180,E1 -21230.232,E2 -21230.232} C_VEL
LIN {X 0,Y 207.168,Z 162.667,A -85,B 0,C 180,E1 -21232.202,E2 -21232.202} C_VEL
LIN {X 0,Y 207.382,Z 162.649,A -85,B 0,C 180,E1 -21238.058,E2 -21238.058} C_VEL
LIN {X 0,Y 207.515,Z 162.631,A -85,B 0,C 180,E1 -21240,E2 -21240} C_VEL
LIN {X 0,Y 207.382,Z 162.643,A -85,B 0,C 180,E1 -21241.943,E2 -21241.943} C_VEL
LIN {X 0,Y 207.167,Z 162.676,A -85,B 0,C 180,E1 -21247.799,E2 -21247.799} C_VEL
LIN {X 0,Y 206.982,Z 162.693,A -85,B 0,C 180,E1 -21251.755,E2 -21251.755} C_VEL
LIN {X 0,Y 206.868,Z 162.715,A -85,B 0,C 180,E1 -21255.771,E2 -21255.771} C_VEL
LIN {X 0,Y 206.763,Z 162.723,A -85,B 0,C 180,E1 -21259.872,E2 -21259.872} C_VEL
LIN {X 0,Y 206.748,Z 162.732,A -85,B 0,C 180,E1 -21264.075,E2 -21264.075} C_VEL
LIN {X 0,Y 206.745,Z 162.732,A -85,B 0,C 180,E1 -21268.419,E2 -21268.419} C_VEL
LIN {X 0,Y 206.71,Z 162.736,A -85,B 0,C 180,E1 -21272.956,E2 -21272.956} C_VEL
LIN {X 0,Y 206.723,Z 162.734,A -85,B 0,C 180,E1 -21275.321,E2 -21275.321} C_VEL
LIN {X 0,Y 206.68,Z 162.739,A -85,B 0,C 180,E1 -21280.247,E2 -21280.247} C_VEL
LIN {X 0,Y 206.685,Z 162.739,A -85,B 0,C 180,E1 -21284.433,E2 -21284.433} C_VEL
LIN {X 0,Y 206.74,Z 162.931,A -85,B 0,C 180,E1 -21289.179,E2 -21289.179} C_VEL
LIN {X 0,Y 208.689,Z 170.986,A -85,B 0,C 180,E1 -21292.825,E2 -21292.825} C_VEL
LIN {X 0,Y 209.087,Z 173.467,A -85,B 0,C 180,E1 -21293.627,E2 -21293.627} C_VEL
LIN {X 0,Y 209.354,Z 176.588,A -85,B 0,C 180,E1 -21294.253,E2 -21294.253} C_VEL
LIN {X 0,Y 209.624,Z 181.97,A -85,B 0,C 180,E1 -21294.925,E2 -21294.925} C_VEL
LIN {X 0,Y 210.898,Z 195.942,A -85,B 0,C 180,E1 -21295.852,E2 -21295.852} C_VEL
LIN {X 0,Y 211.785,Z 199.851,A -85,B 0,C 180,E1 -21296.136,E2 -21296.136} C_VEL
LIN {X 0,Y 214.517,Z 221.54,A -85,B 0,C 180,E1 -21297.389,E2 -21297.389} C_VEL
LIN {X 0,Y 215.93,Z 237.239,A -85,B 0,C 180,E1 -21298.205,E2 -21298.205} C_VEL
LIN {X 0,Y 213.737,Z 284.904,A -85,B 0,C 180,E1 -21299.943,E2 -21299.943} C_VEL
LIN {X 0,Y 212.644,Z 297.116,A -85,B 0,C 180,E1 -21300.688,E2 -21300.688} C_VEL
LIN {X 0,Y 211.036,Z 309.716,A -85,B 0,C 180,E1 -21301.805,E2 -21301.805} C_VEL
LIN {X 0,Y 209.007,Z 321.862,A -85,B 0,C 180,E1 -21303.273,E2 -21303.273} C_VEL
LIN {X 0,Y 207.048,Z 332.152,A -85,B 0,C 180,E1 -21304.894,E2 -21304.894} C_VEL
LIN {X 0,Y 204.731,Z 342.83,A -85,B 0,C 180,E1 -21307.016,E2 -21307.016} C_VEL
LIN {X 0,Y 202.714,Z 352.352,A -85,B 0,C 180,E1 -21309.404,E2 -21309.404} C_VEL
LIN {X 0,Y 201.175,Z 359.682,A -85,B 0,C 180,E1 -21311.675,E2 -21311.675} C_VEL
LIN {X 0,Y 199.547,Z 367.544,A -85,B 0,C 180,E1 -21314.684,E2 -21314.684} C_VEL
LIN {X 0,Y 198.359,Z 373.811,A -85,B 0,C 180,E1 -21317.726,E2 -21317.726} C_VEL
LIN {X 0,Y 197.773,Z 378.771,A -85,B 0,C 180,E1 -21320.798,E2 -21320.798} C_VEL
LIN {X 0,Y 197.575,Z 382.547,A -85,B 0,C 180,E1 -21323.874,E2 -21323.874} C_VEL
LIN {X 0,Y 197.577,Z 384.468,A -85,B 0,C 180,E1 -21325.92,E2 -21325.92} C_VEL
LIN {X 0,Y 197.649,Z 385.932,A -85,B 0,C 180,E1 -21327.962,E2 -21327.962} C_VEL
LIN {X 0,Y 197.685,Z 386.92,A -85,B 0,C 180,E1 -21330,E2 -21330} C_VEL
LIN {X 0,Y 197.588,Z 387.489,A -85,B 0,C 180,E1 -21332.038,E2 -21332.038} C_VEL
LIN {X 0,Y 197.378,Z 387.65,A -85,B 0,C 180,E1 -21334.44,E2 -21334.44} C_VEL
LIN {X 0,Y 197.493,Z 386.752,A -85,B 0,C 180,E1 -21338.183,E2 -21338.183} C_VEL
LIN {X 0,Y 198.426,Z 384.262,A -85,B 0,C 180,E1 -21342.269,E2 -21342.269} C_VEL
LIN {X 0,Y 199.716,Z 381.303,A -85,B 0,C 180,E1 -21345.303,E2 -21345.303} C_VEL
LIN {X 0,Y 201.67,Z 377.357,A -85,B 0,C 180,E1 -21348.279,E2 -21348.279} C_VEL
LIN {X 0,Y 204.151,Z 372.319,A -85,B 0,C 180,E1 -21351.19,E2 -21351.19} C_VEL
LIN {X 0,Y 207.005,Z 366.048,A -85,B 0,C 180,E1 -21354.042,E2 -21354.042} C_VEL
LIN {X 0,Y 210.541,Z 358.319,A -85,B 0,C 180,E1 -21356.784,E2 -21356.784} C_VEL
LIN {X 0,Y 213.88,Z 350.475,A -85,B 0,C 180,E1 -21358.991,E2 -21358.991} C_VEL
LIN {X 0,Y 218.078,Z 339.923,A -85,B 0,C 180,E1 -21361.309,E2 -21361.309} C_VEL
LIN {X 0,Y 221.841,Z 329.303,A -85,B 0,C 180,E1 -21363.126,E2 -21363.126} C_VEL
LIN {X 0,Y 225.401,Z 317.451,A -85,B 0,C 180,E1 -21364.683,E2 -21364.683} C_VEL
LIN {X 0,Y 228.523,Z 304.962,A -85,B 0,C 180,E1 -21365.891,E2 -21365.891} C_VEL
LIN {X 0,Y 230.968,Z 291.975,A -85,B 0,C 180,E1 -21366.802,E2 -21366.802} C_VEL
LIN {X 0,Y 232.518,Z 278.653,A -85,B 0,C 180,E1 -21367.436,E2 -21367.436} C_VEL
LIN {X 0,Y 235.165,Z 240.347,A -85,B 0,C 180,E1 -21368.723,E2 -21368.723} C_VEL
LIN {X 0,Y 233.812,Z 224.78,A -85,B 0,C 180,E1 -21369.909,E2 -21369.909} C_VEL
LIN {X 0,Y 229.811,Z 214.972,A -85,B 0,C 180,E1 -21371.654,E2 -21371.654} C_VEL
LIN {X 0,Y 225.921,Z 206.65,A -85,B 0,C 180,E1 -21373.417,E2 -21373.417} C_VEL
LIN {X 0,Y 221.59,Z 198.515,A -85,B 0,C 180,E1 -21375.544,E2 -21375.544} C_VEL
LIN {X 0,Y 218.419,Z 193.112,A -85,B 0,C 180,E1 -21377.207,E2 -21377.207} C_VEL
LIN {X 0,Y 215.126,Z 187.706,A -85,B 0,C 180,E1 -21379.125,E2 -21379.125} C_VEL
LIN {X 0,Y 211.265,Z 181.714,A -85,B 0,C 180,E1 -21381.629,E2 -21381.629} C_VEL
LIN {X 0,Y 207.505,Z 176.347,A -85,B 0,C 180,E1 -21384.473,E2 -21384.473} C_VEL
LIN {X 0,Y 206.736,Z 175.083,A -85,B 0,C 180,E1 -21385.142,E2 -21385.142} C_VEL
LIN {X 0,Y 201.009,Z 167.183,A -85,B 0,C 180,E1 -21391.441,E2 -21391.441} C_VEL
LIN {X 0,Y 199.852,Z 164.371,A -85,B 0,C 180,E1 -21397.242,E2 -21397.242} C_VEL
LIN {X 0,Y 199.722,Z 163.598,A -85,B 0,C 180,E1 -21399.934,E2 -21399.934} C_VEL
LIN {X 0,Y 199.807,Z 163.589,A -85,B 0,C 180,E1 -21403.656,E2 -21403.656} C_VEL
LIN {X 0,Y 200.068,Z 163.555,A -85,B 0,C 180,E1 -21409.602,E2 -21409.602} C_VEL
LIN {X 0,Y 200.103,Z 163.674,A -85,B 0,C 180,E1 -21410.587,E2 -21410.587} C_VEL
LIN {X 0,Y 200.692,Z 165.62,A -85,B 0,C 180,E1 -21411.821,E2 -21411.821} C_VEL
LIN {X 0,Y 202.491,Z 168.09,A -85,B 0,C 180,E1 -21414.273,E2 -21414.273} C_VEL
LIN {X 0,Y 205.55,Z 169.761,A -85,B 0,C 180,E1 -21417.231,E2 -21417.231} C_VEL
LIN {X 0,Y 207.001,Z 172.589,A -85,B 0,C 180,E1 -21418.662,E2 -21418.662} C_VEL
LIN {X 0,Y 209.819,Z 175.121,A -85,B 0,C 180,E1 -21420.792,E2 -21420.792} C_VEL
LIN {X 0,Y 211.641,Z 178.394,A -85,B 0,C 180,E1 -21422.17,E2 -21422.17} C_VEL
LIN {X 0,Y 213.868,Z 180.744,A -85,B 0,C 180,E1 -21423.591,E2 -21423.591} C_VEL
LIN {X 0,Y 216.438,Z 184.254,A -85,B 0,C 180,E1 -21425.12,E2 -21425.12} C_VEL
LIN {X 0,Y 217.623,Z 185.714,A -85,B 0,C 180,E1 -21425.777,E2 -21425.777} C_VEL
LIN {X 0,Y 221.234,Z 191.114,A -85,B 0,C 180,E1 -21427.716,E2 -21427.716} C_VEL
LIN {X 0,Y 225.926,Z 198.049,A -85,B 0,C 180,E1 -21429.936,E2 -21429.936} C_VEL
LIN {X 0,Y 231.464,Z 207.354,A -85,B 0,C 180,E1 -21432.318,E2 -21432.318} C_VEL
LIN {X 0,Y 236.664,Z 217.46,A -85,B 0,C 180,E1 -21434.395,E2 -21434.395} C_VEL
LIN {X 0,Y 233.168,Z 265.574,A -85,B 0,C 180,E1 -21436.012,E2 -21436.012} C_VEL
LIN {X 0,Y 231.438,Z 278.905,A -85,B 0,C 180,E1 -21436.766,E2 -21436.766} C_VEL
LIN {X 0,Y 229.25,Z 291.564,A -85,B 0,C 180,E1 -21437.852,E2 -21437.852} C_VEL
LIN {X 0,Y 226.527,Z 303.299,A -85,B 0,C 180,E1 -21439.213,E2 -21439.213} C_VEL
LIN {X 0,Y 223.01,Z 315.239,A -85,B 0,C 180,E1 -21440.996,E2 -21440.996} C_VEL
LIN {X 0,Y 219.468,Z 325.642,A -85,B 0,C 180,E1 -21443.048,E2 -21443.048} C_VEL
LIN {X 0,Y 215.605,Z 335.261,A -85,B 0,C 180,E1 -21445.452,E2 -21445.452} C_VEL
LIN {X 0,Y 212.243,Z 342.648,A -85,B 0,C 180,E1 -21447.765,E2 -21447.765} C_VEL
LIN {X 0,Y 209.147,Z 348.994,A -85,B 0,C 180,E1 -21450.268,E2 -21450.268} C_VEL
LIN {X 0,Y 206.222,Z 354.538,A -85,B 0,C 180,E1 -21453.043,E2 -21453.043} C_VEL
LIN {X 0,Y 203.68,Z 358.95,A -85,B 0,C 180,E1 -21455.915,E2 -21455.915} C_VEL
LIN {X 0,Y 201.125,Z 363.087,A -85,B 0,C 180,E1 -21459.759,E2 -21459.759} C_VEL
LIN {X 0,Y 199.78,Z 364.977,A -85,B 0,C 180,E1 -21462.375,E2 -21462.375} C_VEL
LIN {X 0,Y 198.687,Z 366.143,A -85,B 0,C 180,E1 -21465.027,E2 -21465.027} C_VEL
LIN {X 0,Y 197.851,Z 366.642,A -85,B 0,C 180,E1 -21468.24,E2 -21468.24} C_VEL
LIN {X 0,Y 197.383,Z 366.121,A -85,B 0,C 180,E1 -21471.566,E2 -21471.566} C_VEL
LIN {X 0,Y 197.357,Z 364.307,A -85,B 0,C 180,E1 -21475.266,E2 -21475.266} C_VEL
LIN {X 0,Y 197.764,Z 361.548,A -85,B 0,C 180,E1 -21478.527,E2 -21478.527} C_VEL
LIN {X 0,Y 198.393,Z 358.291,A -85,B 0,C 180,E1 -21481.296,E2 -21481.296} C_VEL
LIN {X 0,Y 199.511,Z 352.458,A -85,B 0,C 180,E1 -21484.994,E2 -21484.994} C_VEL
LIN {X 0,Y 201.139,Z 345.165,A -85,B 0,C 180,E1 -21488.477,E2 -21488.477} C_VEL
LIN {X 0,Y 202.821,Z 337.567,A -85,B 0,C 180,E1 -21491.306,E2 -21491.306} C_VEL
LIN {X 0,Y 204.971,Z 328.169,A -85,B 0,C 180,E1 -21494.08,E2 -21494.08} C_VEL
LIN {X 0,Y 207.025,Z 318.084,A -85,B 0,C 180,E1 -21496.463,E2 -21496.463} C_VEL
LIN {X 0,Y 208.962,Z 307.955,A -85,B 0,C 180,E1 -21498.358,E2 -21498.358} C_VEL
LIN {X 0,Y 211.009,Z 295.576,A -85,B 0,C 180,E1 -21500.172,E2 -21500.172} C_VEL
LIN {X 0,Y 212.55,Z 283.214,A -85,B 0,C 180,E1 -21501.554,E2 -21501.554} C_VEL
LIN {X 0,Y 213.85,Z 269.687,A -85,B 0,C 180,E1 -21502.614,E2 -21502.614} C_VEL
LIN {X 0,Y 214.694,Z 256.414,A -85,B 0,C 180,E1 -21503.276,E2 -21503.276} C_VEL
LIN {X 0,Y 217.33,Z 202.011,A -85,B 0,C 180,E1 -21505.175,E2 -21505.175} C_VEL
LIN {X 0,Y 209.697,Z 183.814,A -85,B 0,C 180,E1 -21506.942,E2 -21506.942} C_VEL
LIN {X 0,Y 200.547,Z 164.348,A -85,B 0,C 180,E1 -21509.154,E2 -21509.154} C_VEL
LIN {X 0,Y 200.398,Z 163.524,A -85,B 0,C 180,E1 -21509.247,E2 -21509.247} C_VEL
LIN {X 0,Y 200.319,Z 163.534,A -85,B 0,C 180,E1 -21512.011,E2 -21512.011} C_VEL
LIN {X 0,Y 200.075,Z 163.563,A -85,B 0,C 180,E1 -21518.077,E2 -21518.077} C_VEL
LIN {X 0,Y 199.865,Z 163.589,A -85,B 0,C 180,E1 -21522.18,E2 -21522.18} C_VEL
LIN {X 0,Y 199.766,Z 163.6,A -85,B 0,C 180,E1 -21526.347,E2 -21526.347} C_VEL
LIN {X 0,Y 199.672,Z 163.612,A -85,B 0,C 180,E1 -21530.608,E2 -21530.608} C_VEL
LIN {X 0,Y 199.664,Z 163.614,A -85,B 0,C 180,E1 -21534.985,E2 -21534.985} C_VEL
LIN {X 0,Y 199.674,Z 163.611,A -85,B 0,C 180,E1 -21539.522,E2 -21539.522} C_VEL
LIN {X 0,Y 199.678,Z 163.612,A -85,B 0,C 180,E1 -21542.359,E2 -21542.359} C_VEL
LIN {X 0,Y 199.622,Z 163.619,A -85,B 0,C 180,E1 -21546.763,E2 -21546.763} C_VEL
LIN {X 0,Y 199.608,Z 163.616,A -85,B 0,C 180,E1 -21549.328,E2 -21549.328} C_VEL
LIN {X 0,Y 199.573,Z 163.617,A -85,B 0,C 180,E1 -21552.31,E2 -21552.31} C_VEL
LIN {X 0,Y 199.578,Z 163.623,A -85,B 0,C 180,E1 -21555.229,E2 -21555.229} C_VEL
LIN {X 0,Y 199.637,Z 163.604,A -85,B 0,C 180,E1 -21560.679,E2 -21560.679} C_VEL
LIN {X 0,Y 199.633,Z 163.617,A -85,B 0,C 180,E1 -21565.718,E2 -21565.718} C_VEL
LIN {X 0,Y 199.695,Z 163.603,A -85,B 0,C 180,E1 -21568.136,E2 -21568.136} C_VEL
LIN {X 0,Y 199.684,Z 163.603,A -85,B 0,C 180,E1 -21572.772,E2 -21572.772} C_VEL
LIN {X 0,Y 199.714,Z 163.607,A -85,B 0,C 180,E1 -21577.227,E2 -21577.227} C_VEL
LIN {X 0,Y 199.795,Z 163.581,A -85,B 0,C 180,E1 -21581.759,E2 -21581.759} C_VEL
LIN {X 0,Y 199.848,Z 163.589,A -85,B 0,C 180,E1 -21585.75,E2 -21585.75} C_VEL
LIN {X 0,Y 200.07,Z 163.558,A -85,B 0,C 180,E1 -21589.885,E2 -21589.885} C_VEL
LIN {X 0,Y 200.035,Z 163.552,A -85,B 0,C 180,E1 -21593.95,E2 -21593.95} C_VEL
LIN {X 0,Y 200.322,Z 163.528,A -85,B 0,C 180,E1 -21597.99,E2 -21597.99} C_VEL
LIN {X 0,Y 200.48,Z 163.507,A -85,B 0,C 180,E1 -21600,E2 -21600} C_VEL
LIN {X 0,Y 200.029,Z 163.554,A -85,B 0,C 180,E1 -21604.03,E2 -21604.03} C_VEL
LIN {X 0,Y 200.111,Z 163.555,A -85,B 0,C 180,E1 -21608.076,E2 -21608.076} C_VEL
LIN {X 0,Y 199.914,Z 163.573,A -85,B 0,C 180,E1 -21612.177,E2 -21612.177} C_VEL
LIN {X 0,Y 199.805,Z 163.596,A -85,B 0,C 180,E1 -21616.344,E2 -21616.344} C_VEL
LIN {X 0,Y 199.682,Z 163.605,A -85,B 0,C 180,E1 -21620.608,E2 -21620.608} C_VEL
LIN {X 0,Y 199.665,Z 163.611,A -85,B 0,C 180,E1 -21624.986,E2 -21624.986} C_VEL
LIN {X 0,Y 199.676,Z 163.613,A -85,B 0,C 180,E1 -21629.523,E2 -21629.523} C_VEL
LIN {X 0,Y 199.665,Z 163.612,A -85,B 0,C 180,E1 -21632.353,E2 -21632.353} C_VEL
LIN {X 0,Y 199.641,Z 163.616,A -85,B 0,C 180,E1 -21636.76,E2 -21636.76} C_VEL
LIN {X 0,Y 199.642,Z 163.615,A -85,B 0,C 180,E1 -21639.321,E2 -21639.321} C_VEL
LIN {X 0,Y 199.621,Z 163.618,A -85,B 0,C 180,E1 -21642.325,E2 -21642.325} C_VEL
LIN {X 0,Y 199.632,Z 163.616,A -85,B 0,C 180,E1 -21645.244,E2 -21645.244} C_VEL
LIN {X 0,Y 199.653,Z 163.747,A -85,B 0,C 180,E1 -21648.415,E2 -21648.415} C_VEL
LIN {X 0,Y 201.894,Z 172.997,A -85,B 0,C 180,E1 -21652.752,E2 -21652.752} C_VEL
LIN {X 0,Y 202.374,Z 175.169,A -85,B 0,C 180,E1 -21653.721,E2 -21653.721} C_VEL
LIN {X 0,Y 211.126,Z 198.003,A -85,B 0,C 180,E1 -21655.97,E2 -21655.97} C_VEL
LIN {X 0,Y 211.785,Z 199.851,A -85,B 0,C 180,E1 -21656.136,E2 -21656.136} C_VEL
LIN {X 0,Y 212.409,Z 203.601,A -85,B 0,C 180,E1 -21656.375,E2 -21656.375} C_VEL
LIN {X 0,Y 212.084,Z 209.452,A -85,B 0,C 180,E1 -21656.58,E2 -21656.58} C_VEL
LIN {X 0,Y 208.936,Z 225.212,A -85,B 0,C 180,E1 -21656.844,E2 -21656.844} C_VEL
LIN {X 0,Y 208.949,Z 231.132,A -85,B 0,C 180,E1 -21657.097,E2 -21657.097} C_VEL
LIN {X 0,Y 209.408,Z 238.2,A -85,B 0,C 180,E1 -21657.455,E2 -21657.455} C_VEL
LIN {X 0,Y 207.201,Z 284.441,A -85,B 0,C 180,E1 -21659.194,E2 -21659.194} C_VEL
LIN {X 0,Y 206.098,Z 296.47,A -85,B 0,C 180,E1 -21659.944,E2 -21659.944} C_VEL
LIN {X 0,Y 204.442,Z 309.132,A -85,B 0,C 180,E1 -21661.091,E2 -21661.091} C_VEL
LIN {X 0,Y 202.344,Z 321.335,A -85,B 0,C 180,E1 -21662.599,E2 -21662.599} C_VEL
LIN {X 0,Y 199.963,Z 332.926,A -85,B 0,C 180,E1 -21664.498,E2 -21664.498} C_VEL
LIN {X 0,Y 197.729,Z 343.44,A -85,B 0,C 180,E1 -21666.708,E2 -21666.708} C_VEL
LIN {X 0,Y 195.798,Z 352.043,A -85,B 0,C 180,E1 -21668.965,E2 -21668.965} C_VEL
LIN {X 0,Y 194.365,Z 358.471,A -85,B 0,C 180,E1 -21671.009,E2 -21671.009} C_VEL
LIN {X 0,Y 192.665,Z 366.535,A -85,B 0,C 180,E1 -21674.122,E2 -21674.122} C_VEL
LIN {X 0,Y 191.381,Z 372.925,A -85,B 0,C 180,E1 -21677.271,E2 -21677.271} C_VEL
LIN {X 0,Y 190.717,Z 377.99,A -85,B 0,C 180,E1 -21680.455,E2 -21680.455} C_VEL
LIN {X 0,Y 190.5,Z 381.867,A -85,B 0,C 180,E1 -21683.646,E2 -21683.646} C_VEL
LIN {X 0,Y 190.487,Z 383.835,A -85,B 0,C 180,E1 -21685.768,E2 -21685.768} C_VEL
LIN {X 0,Y 190.582,Z 385.366,A -85,B 0,C 180,E1 -21687.887,E2 -21687.887} C_VEL
LIN {X 0,Y 190.618,Z 386.421,A -85,B 0,C 180,E1 -21690,E2 -21690} C_VEL
LIN {X 0,Y 190.492,Z 387.031,A -85,B 0,C 180,E1 -21692.114,E2 -21692.114} C_VEL
LIN {X 0,Y 190.304,Z 387.237,A -85,B 0,C 180,E1 -21694.343,E2 -21694.343} C_VEL
LIN {X 0,Y 190.452,Z 386.462,A -85,B 0,C 180,E1 -21698.488,E2 -21698.488} C_VEL
LIN {X 0,Y 191.454,Z 384.07,A -85,B 0,C 180,E1 -21702.724,E2 -21702.724} C_VEL
LIN {X 0,Y 192.856,Z 381.216,A -85,B 0,C 180,E1 -21705.861,E2 -21705.861} C_VEL
LIN {X 0,Y 194.899,Z 377.372,A -85,B 0,C 180,E1 -21708.937,E2 -21708.937} C_VEL
LIN {X 0,Y 197.973,Z 371.516,A -85,B 0,C 180,E1 -21712.432,E2 -21712.432} C_VEL
LIN {X 0,Y 201.098,Z 365.156,A -85,B 0,C 180,E1 -21715.348,E2 -21715.348} C_VEL
LIN {X 0,Y 204.933,Z 357.322,A -85,B 0,C 180,E1 -21718.134,E2 -21718.134} C_VEL
LIN {X 0,Y 208.579,Z 349.39,A -85,B 0,C 180,E1 -21720.359,E2 -21720.359} C_VEL
LIN {X 0,Y 212.947,Z 338.734,A -85,B 0,C 180,E1 -21722.713,E2 -21722.713} C_VEL
LIN {X 0,Y 216.886,Z 327.938,A -85,B 0,C 180,E1 -21724.546,E2 -21724.546} C_VEL
LIN {X 0,Y 220.636,Z 315.774,A -85,B 0,C 180,E1 -21726.106,E2 -21726.106} C_VEL
LIN {X 0,Y 223.638,Z 304.042,A -85,B 0,C 180,E1 -21727.225,E2 -21727.225} C_VEL
LIN {X 0,Y 226.175,Z 290.785,A -85,B 0,C 180,E1 -21728.139,E2 -21728.139} C_VEL
LIN {X 0,Y 227.754,Z 277.469,A -85,B 0,C 180,E1 -21728.764,E2 -21728.764} C_VEL
LIN {X 0,Y 230.383,Z 241.635,A -85,B 0,C 180,E1 -21729.983,E2 -21729.983} C_VEL
LIN {X 0,Y 229.393,Z 228.077,A -85,B 0,C 180,E1 -21731.036,E2 -21731.036} C_VEL
LIN {X 0,Y 224.762,Z 216.607,A -85,B 0,C 180,E1 -21733.201,E2 -21733.201} C_VEL
LIN {X 0,Y 220.23,Z 207.239,A -85,B 0,C 180,E1 -21735.482,E2 -21735.482} C_VEL
LIN {X 0,Y 215.669,Z 198.934,A -85,B 0,C 180,E1 -21738.001,E2 -21738.001} C_VEL
LIN {X 0,Y 212.406,Z 193.425,A -85,B 0,C 180,E1 -21740.002,E2 -21740.002} C_VEL
LIN {X 0,Y 208.83,Z 187.682,A -85,B 0,C 180,E1 -21742.499,E2 -21742.499} C_VEL
LIN {X 0,Y 205.354,Z 182.383,A -85,B 0,C 180,E1 -21745.321,E2 -21745.321} C_VEL
LIN {X 0,Y 204.35,Z 181.035,A -85,B 0,C 180,E1 -21746.244,E2 -21746.244} C_VEL
LIN {X 0,Y 199.369,Z 173.669,A -85,B 0,C 180,E1 -21752.247,E2 -21752.247} C_VEL
LIN {X 0,Y 196.656,Z 170.25,A -85,B 0,C 180,E1 -21758.758,E2 -21758.758} C_VEL
LIN {X 0,Y 196.363,Z 169.819,A -85,B 0,C 180,E1 -21761.208,E2 -21761.208} C_VEL
LIN {X 0,Y 198.01,Z 170.388,A -85,B 0,C 180,E1 -21768.742,E2 -21768.742} C_VEL
LIN {X 0,Y 198.733,Z 170.661,A -85,B 0,C 180,E1 -21770.085,E2 -21770.085} C_VEL
LIN {X 0,Y 200.359,Z 174.157,A -85,B 0,C 180,E1 -21772.948,E2 -21772.948} C_VEL
LIN {X 0,Y 202.843,Z 176.072,A -85,B 0,C 180,E1 -21775.777,E2 -21775.777} C_VEL
LIN {X 0,Y 203.827,Z 176.643,A -85,B 0,C 180,E1 -21776.691,E2 -21776.691} C_VEL
LIN {X 0,Y 205.643,Z 179.675,A -85,B 0,C 180,E1 -21778.47,E2 -21778.47} C_VEL
LIN {X 0,Y 207.819,Z 181.859,A -85,B 0,C 180,E1 -21780.206,E2 -21780.206} C_VEL
LIN {X 0,Y 209.974,Z 185.268,A -85,B 0,C 180,E1 -21781.842,E2 -21781.842} C_VEL
LIN {X 0,Y 211.842,Z 187.457,A -85,B 0,C 180,E1 -21783.09,E2 -21783.09} C_VEL
LIN {X 0,Y 214.479,Z 190.938,A -85,B 0,C 180,E1 -21784.717,E2 -21784.717} C_VEL
LIN {X 0,Y 218.178,Z 196.582,A -85,B 0,C 180,E1 -21786.835,E2 -21786.835} C_VEL
LIN {X 0,Y 222.942,Z 203.919,A -85,B 0,C 180,E1 -21789.226,E2 -21789.226} C_VEL
LIN {X 0,Y 228.168,Z 213.028,A -85,B 0,C 180,E1 -21791.612,E2 -21791.612} C_VEL
LIN {X 0,Y 231.859,Z 220.295,A -85,B 0,C 180,E1 -21793.166,E2 -21793.166} C_VEL
LIN {X 0,Y 228.285,Z 266.407,A -85,B 0,C 180,E1 -21794.746,E2 -21794.746} C_VEL
LIN {X 0,Y 226.503,Z 279.464,A -85,B 0,C 180,E1 -21795.502,E2 -21795.502} C_VEL
LIN {X 0,Y 224.213,Z 291.982,A -85,B 0,C 180,E1 -21796.593,E2 -21796.593} C_VEL
LIN {X 0,Y 221.546,Z 303.087,A -85,B 0,C 180,E1 -21797.886,E2 -21797.886} C_VEL
LIN {X 0,Y 218.058,Z 314.539,A -85,B 0,C 180,E1 -21799.586,E2 -21799.586} C_VEL
LIN {X 0,Y 214.694,Z 324.09,A -85,B 0,C 180,E1 -21801.409,E2 -21801.409} C_VEL
LIN {X 0,Y 211.046,Z 333.071,A -85,B 0,C 180,E1 -21803.553,E2 -21803.553} C_VEL
LIN {X 0,Y 206.995,Z 341.736,A -85,B 0,C 180,E1 -21806.192,E2 -21806.192} C_VEL
LIN {X 0,Y 203.414,Z 348.73,A -85,B 0,C 180,E1 -21808.927,E2 -21808.927} C_VEL
LIN {X 0,Y 200.205,Z 354.416,A -85,B 0,C 180,E1 -21811.773,E2 -21811.773} C_VEL
LIN {X 0,Y 197.226,Z 359.279,A -85,B 0,C 180,E1 -21814.957,E2 -21814.957} C_VEL
LIN {X 0,Y 194.389,Z 363.552,A -85,B 0,C 180,E1 -21819.045,E2 -21819.045} C_VEL
LIN {X 0,Y 192.349,Z 366.064,A -85,B 0,C 180,E1 -21823.051,E2 -21823.051} C_VEL
LIN {X 0,Y 190.92,Z 367.038,A -85,B 0,C 180,E1 -21827.41,E2 -21827.41} C_VEL
LIN {X 0,Y 190.323,Z 366.555,A -85,B 0,C 180,E1 -21831.116,E2 -21831.116} C_VEL
LIN {X 0,Y 190.207,Z 365.115,A -85,B 0,C 180,E1 -21834.378,E2 -21834.378} C_VEL
LIN {X 0,Y 190.566,Z 362.353,A -85,B 0,C 180,E1 -21838.019,E2 -21838.019} C_VEL
LIN {X 0,Y 191.421,Z 358.081,A -85,B 0,C 180,E1 -21841.781,E2 -21841.781} C_VEL
LIN {X 0,Y 192.361,Z 353.234,A -85,B 0,C 180,E1 -21844.943,E2 -21844.943} C_VEL
LIN {X 0,Y 193.813,Z 346.851,A -85,B 0,C 180,E1 -21848.181,E2 -21848.181} C_VEL
LIN {X 0,Y 195.523,Z 339.54,A -85,B 0,C 180,E1 -21851.125,E2 -21851.125} C_VEL
LIN {X 0,Y 197.528,Z 331.032,A -85,B 0,C 180,E1 -21853.873,E2 -21853.873} C_VEL
LIN {X 0,Y 199.756,Z 320.662,A -85,B 0,C 180,E1 -21856.521,E2 -21856.521} C_VEL
LIN {X 0,Y 201.99,Z 309.778,A -85,B 0,C 180,E1 -21858.714,E2 -21858.714} C_VEL
LIN {X 0,Y 204.041,Z 297.842,A -85,B 0,C 180,E1 -21860.584,E2 -21860.584} C_VEL
LIN {X 0,Y 205.819,Z 284.668,A -85,B 0,C 180,E1 -21862.15,E2 -21862.15} C_VEL
LIN {X 0,Y 207.178,Z 271.628,A -85,B 0,C 180,E1 -21863.243,E2 -21863.243} C_VEL
LIN {X 0,Y 208.118,Z 258.069,A -85,B 0,C 180,E1 -21863.973,E2 -21863.973} C_VEL
LIN {X 0,Y 210.805,Z 203.558,A -85,B 0,C 180,E1 -21865.945,E2 -21865.945} C_VEL
LIN {X 0,Y 203.579,Z 186.426,A -85,B 0,C 180,E1 -21867.7,E2 -21867.7} C_VEL
LIN {X 0,Y 194.261,Z 166.959,A -85,B 0,C 180,E1 -21870.039,E2 -21870.039} C_VEL
LIN {X 0,Y 193.388,Z 164.396,A -85,B 0,C 180,E1 -21870.325,E2 -21870.325} C_VEL
LIN {X 0,Y 192.966,Z 164.45,A -85,B 0,C 180,E1 -21874.177,E2 -21874.177} C_VEL
LIN {X 0,Y 193.025,Z 164.442,A -85,B 0,C 180,E1 -21878.374,E2 -21878.374} C_VEL
LIN {X 0,Y 192.791,Z 164.471,A -85,B 0,C 180,E1 -21882.634,E2 -21882.634} C_VEL
LIN {X 0,Y 192.719,Z 164.48,A -85,B 0,C 180,E1 -21886.962,E2 -21886.962} C_VEL
LIN {X 0,Y 192.609,Z 164.491,A -85,B 0,C 180,E1 -21891.4,E2 -21891.4} C_VEL
LIN {X 0,Y 192.647,Z 164.486,A -85,B 0,C 180,E1 -21894.213,E2 -21894.213} C_VEL
LIN {X 0,Y 192.65,Z 164.488,A -85,B 0,C 180,E1 -21898.892,E2 -21898.892} C_VEL
LIN {X 0,Y 192.599,Z 164.493,A -85,B 0,C 180,E1 -21903.186,E2 -21903.186} C_VEL
LIN {X 0,Y 192.551,Z 164.498,A -85,B 0,C 180,E1 -21908.352,E2 -21908.352} C_VEL
LIN {X 0,Y 192.49,Z 164.503,A -85,B 0,C 180,E1 -21913.096,E2 -21913.096} C_VEL
LIN {X 0,Y 192.49,Z 164.504,A -85,B 0,C 180,E1 -21916.904,E2 -21916.904} C_VEL
LIN {X 0,Y 192.573,Z 164.485,A -85,B 0,C 180,E1 -21921.654,E2 -21921.654} C_VEL
LIN {X 0,Y 192.597,Z 164.494,A -85,B 0,C 180,E1 -21924.279,E2 -21924.279} C_VEL
LIN {X 0,Y 192.599,Z 164.483,A -85,B 0,C 180,E1 -21929.279,E2 -21929.279} C_VEL
LIN {X 0,Y 192.66,Z 164.47,A -85,B 0,C 180,E1 -21931.692,E2 -21931.692} C_VEL
LIN {X 0,Y 192.685,Z 164.482,A -85,B 0,C 180,E1 -21936.346,E2 -21936.346} C_VEL
LIN {X 0,Y 192.73,Z 164.461,A -85,B 0,C 180,E1 -21941.459,E2 -21941.459} C_VEL
LIN {X 0,Y 192.772,Z 164.466,A -85,B 0,C 180,E1 -21945.215,E2 -21945.215} C_VEL
LIN {X 0,Y 192.981,Z 164.443,A -85,B 0,C 180,E1 -21949.509,E2 -21949.509} C_VEL
LIN {X 0,Y 193.062,Z 164.424,A -85,B 0,C 180,E1 -21951.628,E2 -21951.628} C_VEL
LIN {X 0,Y 193.264,Z 164.407,A -85,B 0,C 180,E1 -21957.916,E2 -21957.916} C_VEL
LIN {X 0,Y 193.443,Z 164.384,A -85,B 0,C 180,E1 -21960,E2 -21960} C_VEL
LIN {X 0,Y 192.976,Z 164.432,A -85,B 0,C 180,E1 -21964.177,E2 -21964.177} C_VEL
LIN {X 0,Y 193.062,Z 164.434,A -85,B 0,C 180,E1 -21968.373,E2 -21968.373} C_VEL
LIN {X 0,Y 192.853,Z 164.451,A -85,B 0,C 180,E1 -21972.63,E2 -21972.63} C_VEL
LIN {X 0,Y 192.758,Z 164.474,A -85,B 0,C 180,E1 -21976.959,E2 -21976.959} C_VEL
LIN {X 0,Y 192.617,Z 164.488,A -85,B 0,C 180,E1 -21981.4,E2 -21981.4} C_VEL
LIN {X 0,Y 192.648,Z 164.489,A -85,B 0,C 180,E1 -21984.214,E2 -21984.214} C_VEL
LIN {X 0,Y 192.651,Z 164.489,A -85,B 0,C 180,E1 -21988.893,E2 -21988.893} C_VEL
LIN {X 0,Y 192.602,Z 164.493,A -85,B 0,C 180,E1 -21993.186,E2 -21993.186} C_VEL
LIN {X 0,Y 192.611,Z 164.493,A -85,B 0,C 180,E1 -21996.608,E2 -21996.608} C_VEL
LIN {X 0,Y 192.549,Z 164.501,A -85,B 0,C 180,E1 -22001.072,E2 -22001.072} C_VEL
LIN {X 0,Y 192.555,Z 164.501,A -85,B 0,C 180,E1 -22006.095,E2 -22006.095} C_VEL
LIN {X 0,Y 192.611,Z 164.625,A -85,B 0,C 180,E1 -22007.643,E2 -22007.643} C_VEL
LIN {X 0,Y 195.005,Z 174.622,A -85,B 0,C 180,E1 -22012.509,E2 -22012.509} C_VEL
LIN {X 0,Y 202.516,Z 193.824,A -85,B 0,C 180,E1 -22014.587,E2 -22014.587} C_VEL
LIN {X 0,Y 205.892,Z 203.299,A -85,B 0,C 180,E1 -22015.49,E2 -22015.49} C_VEL
LIN {X 0,Y 208.949,Z 231.132,A -85,B 0,C 180,E1 -22017.097,E2 -22017.097} C_VEL
LIN {X 0,Y 208.806,Z 234.37,A -85,B 0,C 180,E1 -22017.217,E2 -22017.217} C_VEL
LIN {X 0,Y 207.274,Z 238.789,A -85,B 0,C 180,E1 -22017.211,E2 -22017.211} C_VEL
LIN {X 0,Y 203.144,Z 247.434,A -85,B 0,C 180,E1 -22017.055,E2 -22017.055} C_VEL
LIN {X 0,Y 202.405,Z 251.4,A -85,B 0,C 180,E1 -22017.132,E2 -22017.132} C_VEL
LIN {X 0,Y 200.634,Z 284.933,A -85,B 0,C 180,E1 -22018.45,E2 -22018.45} C_VEL
LIN {X 0,Y 199.49,Z 296.553,A -85,B 0,C 180,E1 -22019.207,E2 -22019.207} C_VEL
LIN {X 0,Y 197.879,Z 308.547,A -85,B 0,C 180,E1 -22020.33,E2 -22020.33} C_VEL
LIN {X 0,Y 195.721,Z 320.81,A -85,B 0,C 180,E1 -22021.882,E2 -22021.882} C_VEL
LIN {X 0,Y 193.266,Z 332.429,A -85,B 0,C 180,E1 -22023.838,E2 -22023.838} C_VEL
LIN {X 0,Y 190.926,Z 342.958,A -85,B 0,C 180,E1 -22026.114,E2 -22026.114} C_VEL
LIN {X 0,Y 188.76,Z 352.176,A -85,B 0,C 180,E1 -22028.626,E2 -22028.626} C_VEL
LIN {X 0,Y 186.922,Z 360.211,A -85,B 0,C 180,E1 -22031.362,E2 -22031.362} C_VEL
LIN {X 0,Y 185.258,Z 367.808,A -85,B 0,C 180,E1 -22034.6,E2 -22034.6} C_VEL
LIN {X 0,Y 184.111,Z 373.883,A -85,B 0,C 180,E1 -22037.881,E2 -22037.881} C_VEL
LIN {X 0,Y 183.544,Z 378.657,A -85,B 0,C 180,E1 -22041.19,E2 -22041.19} C_VEL
LIN {X 0,Y 183.428,Z 382.714,A -85,B 0,C 180,E1 -22044.998,E2 -22044.998} C_VEL
LIN {X 0,Y 183.492,Z 384.779,A -85,B 0,C 180,E1 -22047.805,E2 -22047.805} C_VEL
LIN {X 0,Y 183.551,Z 385.916,A -85,B 0,C 180,E1 -22050,E2 -22050} C_VEL
LIN {X 0,Y 183.4,Z 386.57,A -85,B 0,C 180,E1 -22052.196,E2 -22052.196} C_VEL
LIN {X 0,Y 183.229,Z 386.817,A -85,B 0,C 180,E1 -22054.4,E2 -22054.4} C_VEL
LIN {X 0,Y 183.402,Z 386.159,A -85,B 0,C 180,E1 -22058.817,E2 -22058.817} C_VEL
LIN {X 0,Y 183.841,Z 385.226,A -85,B 0,C 180,E1 -22061.019,E2 -22061.019} C_VEL
LIN {X 0,Y 185.387,Z 382.147,A -85,B 0,C 180,E1 -22065.389,E2 -22065.389} C_VEL
LIN {X 0,Y 187.43,Z 378.737,A -85,B 0,C 180,E1 -22068.585,E2 -22068.585} C_VEL
LIN {X 0,Y 190.603,Z 373.237,A -85,B 0,C 180,E1 -22072.368,E2 -22072.368} C_VEL
LIN {X 0,Y 194.123,Z 366.602,A -85,B 0,C 180,E1 -22075.75,E2 -22075.75} C_VEL
LIN {X 0,Y 198.003,Z 359.199,A -85,B 0,C 180,E1 -22078.631,E2 -22078.631} C_VEL
LIN {X 0,Y 202.523,Z 350.087,A -85,B 0,C 180,E1 -22081.368,E2 -22081.368} C_VEL
LIN {X 0,Y 207.054,Z 339.675,A -85,B 0,C 180,E1 -22083.766,E2 -22083.766} C_VEL
LIN {X 0,Y 211.616,Z 327.915,A -85,B 0,C 180,E1 -22085.827,E2 -22085.827} C_VEL
LIN {X 0,Y 215.518,Z 315.932,A -85,B 0,C 180,E1 -22087.398,E2 -22087.398} C_VEL
LIN {X 0,Y 218.888,Z 303.334,A -85,B 0,C 180,E1 -22088.615,E2 -22088.615} C_VEL
LIN {X 0,Y 221.463,Z 290.283,A -85,B 0,C 180,E1 -22089.522,E2 -22089.522} C_VEL
LIN {X 0,Y 223.108,Z 277.314,A -85,B 0,C 180,E1 -22090.129,E2 -22090.129} C_VEL
LIN {X 0,Y 225.768,Z 242.268,A -85,B 0,C 180,E1 -22091.345,E2 -22091.345} C_VEL
LIN {X 0,Y 224.926,Z 231.099,A -85,B 0,C 180,E1 -22092.269,E2 -22092.269} C_VEL
LIN {X 0,Y 220.628,Z 220.179,A -85,B 0,C 180,E1 -22094.466,E2 -22094.466} C_VEL
LIN {X 0,Y 216.981,Z 212.455,A -85,B 0,C 180,E1 -22096.418,E2 -22096.418} C_VEL
LIN {X 0,Y 212.972,Z 204.776,A -85,B 0,C 180,E1 -22098.803,E2 -22098.803} C_VEL
LIN {X 0,Y 209.809,Z 199.288,A -85,B 0,C 180,E1 -22100.865,E2 -22100.865} C_VEL
LIN {X 0,Y 206.63,Z 193.904,A -85,B 0,C 180,E1 -22103.247,E2 -22103.247} C_VEL
LIN {X 0,Y 203.345,Z 188.559,A -85,B 0,C 180,E1 -22106.126,E2 -22106.126} C_VEL
LIN {X 0,Y 199.157,Z 182.739,A -85,B 0,C 180,E1 -22110.856,E2 -22110.856} C_VEL
LIN {X 0,Y 197.95,Z 180.422,A -85,B 0,C 180,E1 -22112.799,E2 -22112.799} C_VEL
LIN {X 0,Y 195.57,Z 177.184,A -85,B 0,C 180,E1 -22119.12,E2 -22119.12} C_VEL
LIN {X 0,Y 195.38,Z 176.858,A -85,B 0,C 180,E1 -22123.275,E2 -22123.275} C_VEL
LIN {X 0,Y 197.462,Z 177.658,A -85,B 0,C 180,E1 -22129.684,E2 -22129.684} C_VEL
LIN {X 0,Y 198.978,Z 180.932,A -85,B 0,C 180,E1 -22132.516,E2 -22132.516} C_VEL
LIN {X 0,Y 201.474,Z 182.981,A -85,B 0,C 180,E1 -22135.498,E2 -22135.498} C_VEL
LIN {X 0,Y 202.174,Z 183.463,A -85,B 0,C 180,E1 -22136.179,E2 -22136.179} C_VEL
LIN {X 0,Y 204.199,Z 186.595,A -85,B 0,C 180,E1 -22138.189,E2 -22138.189} C_VEL
LIN {X 0,Y 205.826,Z 188.415,A -85,B 0,C 180,E1 -22139.575,E2 -22139.575} C_VEL
LIN {X 0,Y 208.256,Z 192.09,A -85,B 0,C 180,E1 -22141.473,E2 -22141.473} C_VEL
LIN {X 0,Y 209.685,Z 193.892,A -85,B 0,C 180,E1 -22142.473,E2 -22142.473} C_VEL
LIN {X 0,Y 212.8,Z 198.313,A -85,B 0,C 180,E1 -22144.498,E2 -22144.498} C_VEL
LIN {X 0,Y 217.449,Z 205.585,A -85,B 0,C 180,E1 -22147.182,E2 -22147.182} C_VEL
LIN {X 0,Y 222.046,Z 213.321,A -85,B 0,C 180,E1 -22149.509,E2 -22149.509} C_VEL
LIN {X 0,Y 226.781,Z 222.423,A -85,B 0,C 180,E1 -22151.72,E2 -22151.72} C_VEL
LIN {X 0,Y 227.138,Z 223.219,A -85,B 0,C 180,E1 -22151.881,E2 -22151.881} C_VEL
LIN {X 0,Y 223.614,Z 266.949,A -85,B 0,C 180,E1 -22153.403,E2 -22153.403} C_VEL
LIN {X 0,Y 221.635,Z 280.679,A -85,B 0,C 180,E1 -22154.211,E2 -22154.211} C_VEL
LIN {X 0,Y 219.309,Z 292.655,A -85,B 0,C 180,E1 -22155.279,E2 -22155.279} C_VEL
LIN {X 0,Y 216.398,Z 304.08,A -85,B 0,C 180,E1 -22156.642,E2 -22156.642} C_VEL
LIN {X 0,Y 213.003,Z 314.676,A -85,B 0,C 180,E1 -22158.242,E2 -22158.242} C_VEL
LIN {X 0,Y 208.982,Z 325.388,A -85,B 0,C 180,E1 -22160.325,E2 -22160.325} C_VEL
LIN {X 0,Y 204.784,Z 334.967,A -85,B 0,C 180,E1 -22162.733,E2 -22162.733} C_VEL
LIN {X 0,Y 200.496,Z 343.555,A -85,B 0,C 180,E1 -22165.497,E2 -22165.497} C_VEL
LIN {X 0,Y 196.221,Z 351.168,A -85,B 0,C 180,E1 -22168.731,E2 -22168.731} C_VEL
LIN {X 0,Y 193.134,Z 356.219,A -85,B 0,C 180,E1 -22171.543,E2 -22171.543} C_VEL
LIN {X 0,Y 189.683,Z 361.338,A -85,B 0,C 180,E1 -22175.401,E2 -22175.401} C_VEL
LIN {X 0,Y 186.831,Z 365.075,A -85,B 0,C 180,E1 -22179.753,E2 -22179.753} C_VEL
LIN {X 0,Y 184.915,Z 366.958,A -85,B 0,C 180,E1 -22183.77,E2 -22183.77} C_VEL
